// SIMATIC STEP 7 (V5.x) project COB#1&2_EL#2_01_07_2014
// CPU: CPU 315-2 DP
// CPU: CPU 315-2 DP

SYMBOL_TABLE
"FWD_END_POSI"	DB 1	DB 1	// FWD END POSITION LIMIT SWITCH
"OUTPUT_MAPPING_DB"	DB 2	DB 2	// TRAVEL DELAY TIME
"TRAVEL_DRIVE_DB"	DB 3	DB 3	// QUNCHING START PB
"COMMON_DB"	DB 4	DB 4
"TATA_COMMUNICATION_DB"	DB 5	DB 5	// TATA COMMUNIATION DATA BLOCK
"WinCC_Interface_DB"	DB 6	DB 6
"POWER_ON_DB"	DB 7	DB 7
"ACTUAL_TIME_DB"	DB 8	DB 8
"COMPRESSOR_DB"	DB 9	DB 9
"PROFIBUS_DATA"	DB 10	DB 10
"CMD_FROM_TATA"	DB 11	DB 11	// COMMANDS FROM TATA THROUGH PROFIBUS
"FB_TO_TATA"	DB 12	DB 12	// FEEDBACK TO TATA THROUGH PROFIBUS
"FLAPPER_GATE_DB"	DB 13	DB 13	// FLAPPER GATE DATA BLOCK
"RECEIVE_DB_342-5"	DB 21	DB 21
"SEND_DB_342-5"	DB 22	DB 22
"SPARE_1_DB"	DB 89	DB 89
"SPARE_2_DB"	DB 90	DB 90
"TDISCON"	FB 66	FB 66	// Disconnect
"POWER ON"	FC 2	FC 2	// MAIN POWER ON
"COMPRESSOR"	FC 3	FC 3
"FLAPPER_GATE"	FC 4	FC 4	// FLAPPER GATE FEEDBACKS
"ALARMS"	FC 5	FC 5
"INPUT_MAPPING"	FC 6	FC 6
"OUTPUT_MAPPING"	FC 7	FC 7
"TRAVEL_DRIVE_PROFI_MODE"	FC 8	FC 8
"TRAVEL_DRIVE"	FC 9	FC 9	// TRAVEL DRIVE IN HARDWARE AND PROFIBUS MODES
"PROFIBUS_COMMUNICATION"	FC 10	FC 10	// PROFIBUS COMMUNICATION
"TATA_COMMUNICATION"	FC 11	FC 11	// COMMUNICATION WITH TATA THROUGH PROFIBUS
"FAULT TRAP"	FC 12	FC 12	// FAULT EXAMINATION FC
"SCALE"	FC 105	FC 105	// Scaling Values
"UNSCALE"	FC 106	FC 106	// Unscaling Values
"MAIN PWR RUNG FB"	I 0.0	BOOL	// MAIN POWER RUNNING FEEDBACK
"CONTROL PWR ON FB"	I 0.1	BOOL	// CONTROL POWER ON FEEDBACK
"EMER STOP PB AT CD"	I 0.2	BOOL	// EMERGENCY STOP PUSH BUTTON AT CD
"LAMP TEST PB ATCD"	I 0.3	BOOL	// LAMP TEST PUSH BUTTON AT CD
"ALARM ACK PB AT CD"	I 0.4	BOOL	// ALARM ACKNOWLEDGE PUSH BUTTON AT CD
"MANUAL MODE"	I 0.5	BOOL	// MANUAL MODE SELECTION
"AUTO MODE"	I 0.6	BOOL	// AUTO MODE SELECTION
"LT_CRIPPING_SPEED"	I 0.7	BOOL	// LT TRAVEL CRIPPING SPEED
"PROFIBUS/HW DRV1 SELCT"	I 1.0	BOOL	// PROFIBUS/HARDWARE MODE SELECT DRIVE 1
"TRVL DRV 1 RDY TO START"	I 1.1	BOOL	// TRAVEL DRIVE 1 READY TO START
"TRVL DRV 1 RNG FB"	I 1.2	BOOL	// TRAVEL DRIVE 1 RUNNING FEED BACK
"TRVL DRV 1 OLR TRIP"	I 1.3	BOOL	// TRAVEL DRIVE 1 OLR TRIPPED FEED BACK
"PROFIBUS/HW DRV2 SELCT"	I 1.4	BOOL	// PROFIBUS/HARDWARE MODE SELECT DRIVE 2
"TRVL DRV 2 RDY TO START"	I 1.5	BOOL	// TRAVEL DRIVE 2 READY TO START
"TRVL DRV 2 RNG FB"	I 1.6	BOOL	// TRAVEL DRIVE 2 RUNNING FEED BACK
"TRVL DRV 2 OLR TRIP"	I 1.7	BOOL	// TRAVEL DRIVE 2 OLR TRIPPED FEED BACK
"SPARE _2"	I 2.0	BOOL	// SPARE 2
"SPARE_3"	I 2.1	BOOL	// SPARE_3
"JOY ST DEADMAN BUTTON"	I 2.2	BOOL	// JOYSTICK DEADMAN BUTTON
"JOY ST HOME POS"	I 2.3	BOOL	// JOYSTICK HOME POSITION
"JOY ST FWD POS"	I 2.4	BOOL	// JOYSTICK FORWARD POSITION
"JOY ST REV POS"	I 2.5	BOOL	// JOYSTICK REVERSE POSITION
"EMER STOP AT MCC"	I 2.6	BOOL	// EMERGENCY STOP PUSH BUTTON AT MCC
"QL_NOT_RDY_INPUT"	I 2.7	BOOL	// QUENCHING NOT READY
"FWD END LMT SW FB"	I 3.0	BOOL	// FORWARD END LIMIT SWITCH FEED BACK
"FWD EMER END LMT SW FB"	I 3.1	BOOL	// FORWARD EMERGENCY END LIMIT SWITCH FEED BACK
"REV END LMT SW FB"	I 3.2	BOOL	// REVERSE END LIMIT SWITCH FEED BACK
"REV EMER END LMT SW FB"	I 3.3	BOOL	// REVERSE EMERGENCY END LIMIT SWITCH FEED BACK
"LS_FLAPPER_GATE_1_FB"	I 3.4	BOOL	// LS_FLAPPER_GATE 1 FB
"LS_FLAPPER_GATE_2_FB"	I 3.5	BOOL	// LS FLAPPER GATE 2 FB
"DRIVE_1_ISU_CHARGE"	I 3.6	BOOL	// DRIVE 1 ISU CHARGE
"DRIVE_2_ISU_CHARGE"	I 3.7	BOOL	// DRIVE 2 ISU CHARGE
"COMP 1 RDY TO START"	I 4.0	BOOL	// COMPRESSOR 1 READY TO START PUSH BUTTON
"COMP1 RUNG FB"	I 4.1	BOOL	// COMPRESSOR 1 RUNNING FEED BACK
"COMP 2 RDY TO START"	I 4.2	BOOL	// COMPRESSOR 2 READY TO START PUSH BUTTON
"COMP2 RUNG FB"	I 4.3	BOOL	// COMPRESSOR 2 RUNNING FEED BACK
"COMP 1 & 2 SELECT"	I 4.4	BOOL	// COMPRESSOR 1 & 2 SELECTION
"COMP 1 START PB"	I 4.5	BOOL	// COMPRESSOR 1 START PUSH BUTTON
"COMP 1 STOP PB"	I 4.6	BOOL	// COMPRESSOR 1 STOP PUSH BUTTON
"CD_PC_SEL"	I 4.7	BOOL	// CD OR PC SELECTION SWITCH
"COMP 2 START PB"	I 5.0	BOOL	// COMPRESSOR 2 START PUSH BUTTON
"COMP 2 STOP PB"	I 5.1	BOOL	// COMPRESSOR 2 STOP PUSH BUTTON
"COMP1 MAX PSW FB"	I 5.2	BOOL	// COMPRESSOR 1 MAX PRESSURE SWITCH FEED BACK
"COMP MINI PSW FB"	I 5.3	BOOL	// MINIMUM PRESSURE SWITCH FEED BACK TRAVEL
"COMP BRK LINE PSW FB"	I 5.4	BOOL	// LT BRAKE LINE PRESSURE SWITCH FEED BACK
"COMP2 CNTRL PSW FB"	I 5.5	BOOL	// COMPRESSOR 2 CONTROL PRESSURE SWITCH FEED BACK
"SPARE 4"	I 5.6	BOOL	// SPARE INPUT 4 (I5.6)
"SPARE 5"	I 5.7	BOOL	// SPARE INPUT 5 (I5.7)
"SPARE 6"	I 6.0	BOOL	// SPARE INPUT 6 (I6.0)
"PUSHING_PERMISION"	I 6.1	BOOL	// PUSHING PERMISSION SIGNAL
"FED_END_POSI"	I 6.2	BOOL	// FWD END POSITION LIMIT SWITCH
"SPARE 9"	I 6.3	BOOL	// SPARE INPUT 9 (I6.3)
"SPARE 10"	I 6.4	BOOL	// SPARE INPUT 10 (I6.4)
"SPARE 11"	I 6.5	BOOL	// SPARE INPUT 11 (I6.5)
"SPARE 12"	I 6.6	BOOL	// SPARE INPUT 12 (I6.6)
"SPARE 13"	I 6.7	BOOL	// SPARE INPUT 13 (I6.7)
"SPARE 14"	I 7.0	BOOL	// SPARE INPUT 14 (I7.0)
"SPARE 15"	I 7.1	BOOL	// SPARE INPUT 15 (I7.1)
"SPARE 16"	I 7.2	BOOL	// SPARE INPUT 16 (I7.2)
"SPARE 17"	I 7.3	BOOL	// SPARE INPUT 17 (I7.3)
"SPARE 18"	I 7.4	BOOL	// SPARE INPUT 18 (I7.4)
"SPARE 19"	I 7.5	BOOL	// SPARE INPUT 19 (I7.5)
"SPARE 20"	I 7.6	BOOL	// SPARE INPUT 20 (I7.6)
"SPARE 21"	I 7.7	BOOL	// SPARE INPUT 21 (I7.7)
"LOW BIT"	M 0.0	BOOL	// ALWAYS LOW BIT
"HIGH BIT"	M 0.1	BOOL	// ALWAYS HIGH BIT
"QUENCHING_INPUT_LS"	M 2.0	BOOL
"40S_LT_ON_DELAY"	M 2.1	BOOL	// 40 SECOND LT ON DELAY
"QUEN_DELEY_TIME"	M 2.2	BOOL	// QIENCHING DELAY OFF TIME
"LT_PERMISSION"	M 2.3	BOOL	// LT  AFTER QUENCHING PERMISSION
"COMP_1_RDY_2_STRT_FLT"	M 2.4	BOOL	// COMP#1 READY TO START FEEDBACK FAULT
"EMER_CD_FLT"	M 2.5	BOOL	// EMERGENCY AT CD FAULT
"COMP_1_STP_PB_FLT"	M 2.6	BOOL	// COMP#1 STOP PUSH BUTTON FAULT
"COMP_2_RDY_FR_STRT_FLT"	M 2.7	BOOL	// COMPRESSOR 2 READY FOR START FAULT
"COMP_2_OFF_PB_FLT"	M 3.0	BOOL	// COMPRESSOR 2 OFF PUSH BUTTON FAULT
"RESET FAULTS"	M 3.1	BOOL	// RESET ALL FAULTS
"COMP_SELEC_SW_FLT"	M 3.2	BOOL	// COMPRESSOR SELECTOR SWITCH FAULT
"MAIN_PWR_FLT"	M 3.3	BOOL	// MAIN POWER ON FEEDBACK FAULT
"CTRL_PWR_FLT"	M 3.4	BOOL	// CONTROL POWER ON FEEDBACK FAULT
"CYCLIC_EXECUCTION"	OB 1	OB 1	// Cycle Execution
"CYCL_FLT"	OB 80	OB 80	// Cycle Time Fault
"I/O_FLT1"	OB 82	OB 82	// I/O Point Fault 1
"OBNL_FLT"	OB 85	OB 85	// OB Not Loaded Fault
"RACK_FLT"	OB 86	OB 86	// Loss of Rack Fault
"COMM_FLT"	OB 87	OB 87	// Communication Fault
"COMPLETE RESTART"	OB 100	OB 100	// Complete Restart
"PROG_ERR"	OB 121	OB 121	// Programming Error
"MOD_ERR"	OB 122	OB 122	// Module Access Error
"JOY_STICK_SPEED_REF"	PIW 254	INT	// SPEED REFERENCE FROM JOY STICK
"SPEED_REF_TO_DRV_1"	PQW 258	INT	// SPEED REFERENCE TO TRAVEL DRIVE 1
"SPEED_REF_TO_DRV_2"	PQW 260	INT	// SPEED REFERENCE TO TRAVEL DRIVE 2
"CNTRL_ PWR_ ON_ IND"	Q 0.2	BOOL	// CONTROL POWER ON INDICATION
"COMP_ 1_ON_CMD"	Q 0.3	BOOL	// COMPRESSOR-1 ON COMMAND
"COMP_ 2_ON_CMD"	Q 0.4	BOOL	// COMPRESSOR 2 ON COMMAND
"FLAPPER_GATE_1_POSITION"	Q 0.5	BOOL	// FLAPPER_GATE_1_POSITION
"FLAPPER_GATE_2_POSITION"	Q 0.6	BOOL	// "FLAPPER_GATE_2_POSITION"
"FLAP_GATE_1_OPN_IND"	Q 0.7	BOOL	// FLAPPER GATE 1 OPEN INDICATION
"TRA_DRIVE_1_FWD_COM"	Q 1.0	BOOL	// TRAVEL DRIVE 1 FORWARD COMMAND
"TRA_DRIVE_1_REV_COM"	Q 1.1	BOOL	// TRAVEL DRIVE 1 REVERSE COMMAND
"TRA_DRIVE_2_FWD_COM"	Q 1.2	BOOL	// TRAVEL DRIVE 2 FORWRD COMMAND
"TRA_DRIVE_2_REV_COM"	Q 1.3	BOOL	// TRAVEL DRIVE 2 REVERSE COMMAND
"COM_1_ON_IND"	Q 1.4	BOOL	// COMPRESSOR 1 ON INDICATION
"COM_2_ON_IND"	Q 1.5	BOOL	// COMPRESSOR 2 ON INDICATION
"TRA_PERMISSION_IND"	Q 1.6	BOOL	// TRAVEL PERMISSION INDICATION
"FLAP_GATE_2_OPN_IND"	Q 1.7	BOOL	// FLAPPER GATE 2 OPEN INDICATION
"DRV_1_ISU_CMD"	Q 2.0	BOOL	// DRIVE 1 ISU CHARGE COMMAND
"DRV_2_ISU_CMD"	Q 2.1	BOOL	// DRIVE 2 ISU CHARGE COMMAND
"LIGHT_ON_CMD"	Q 2.2	BOOL	// LIGHT ON COMMAND
"SPARE_12"	Q 2.3	BOOL	// SPARE_12
"SPARE OP 9"	Q 2.4	BOOL	// SPARE OUPUT 1 (Q2.4)
"SPARE OP 10"	Q 2.5	BOOL	// TRAVEL DELAY TIME (Q2.5)
"SPARE OP 11"	Q 2.6	BOOL	// SPARE OUPUT 1 (Q2.6)
"SPARE OP 12"	Q 2.7	BOOL	// SPARE OUPUT 1 (Q2.7)
"SPARE OP 13"	Q 3.0	BOOL	// SPARE OUPUT 1 (Q3.0)
"SPARE OP 14"	Q 3.1	BOOL	// SPARE OUPUT 1 (Q3.1)
"SPARE OP 15"	Q 3.2	BOOL	// SPARE OUPUT 1 (Q3.2)
"SPARE OP 16"	Q 3.3	BOOL	// SPARE OUPUT 1 (Q3.3)
"SPARE OP 17"	Q 3.4	BOOL	// SPARE OUPUT 1 (Q3.4)
"SPARE OP 18"	Q 3.5	BOOL	// SPARE OUPUT 1 (Q3.5)
"SPARE OP 19"	Q 3.6	BOOL	// SPARE OUPUT 1 (Q3.6)
"SPARE OP 20"	Q 3.7	BOOL	// SPARE OUPUT 1 (Q3.7)
"HOOTER_ON_OP"	Q 4.0	BOOL	// HOOTER ON OUTPUT
"DPRD_DAT"	SFC 14	SFC 14	// Read Consistent Data of a Standard DP Slave
"DPWR_DAT"	SFC 15	SFC 15	// Write Consistent Data to a Standard DP Slave
"VAT_1"	VAT 1	
"FAULT_EXAMINATION"	VAT 2		// FAULT EXAMINATION TABLE
"LOCO#2_FORCE TABLE"	VAT 3	
END_SYMBOL_TABLE

// FB 66: know-how protected block, not included

FUNCTION "POWER ON" : VOID	// FC 2
VERSION : 0.1
VAR_TEMP
  TEMP0 : WORD ;
  TEMP1 : WORD ;
  TEMP2 : WORD ;
END_VAR
BEGIN
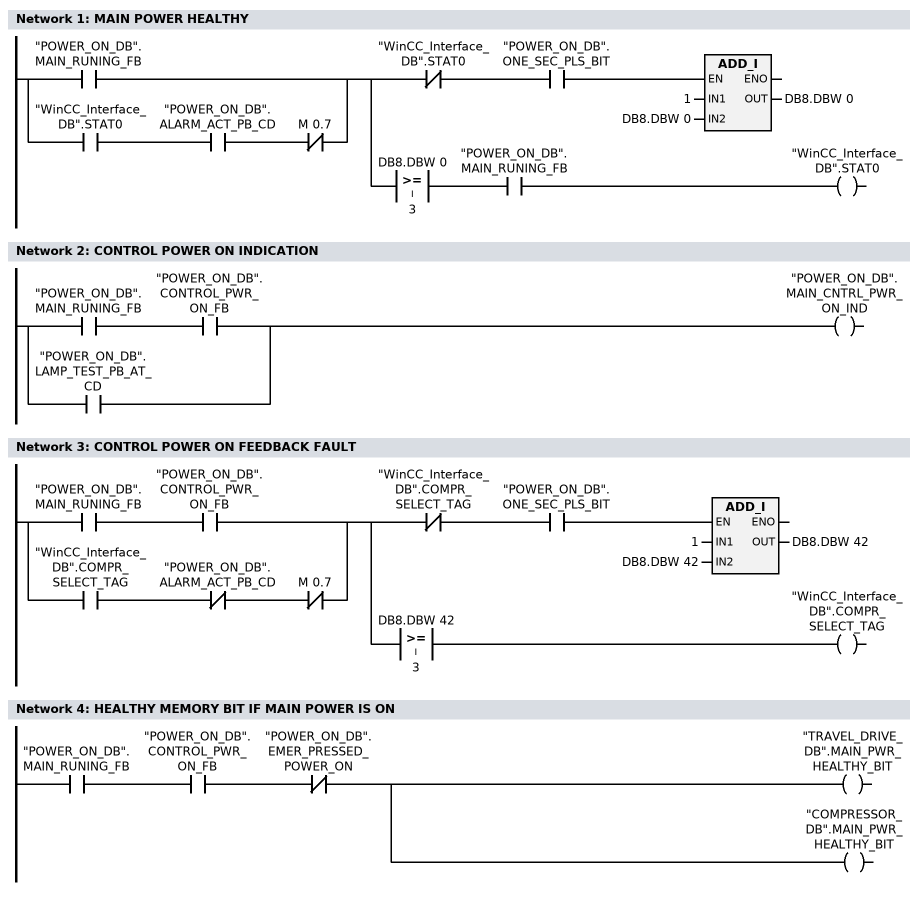
NETWORK
TITLE = MAIN POWER HEALTHY
      O     "POWER_ON_DB".MAIN_RUNING_FB;
      O;
      A     "WinCC_Interface_DB".STAT0;
      A     "POWER_ON_DB".ALARM_ACT_PB_CD;
      AN    M 0.7;
      =     L 6.0;
      A     L 6.0;
      AN    "WinCC_Interface_DB".STAT0;
      A     "POWER_ON_DB".ONE_SEC_PLS_BIT;
      JNB   _001;
      L     1;
      L     DB8.DBW 0;
      +I;
      T     DB8.DBW 0;
_001: NOP   0;
      A     L 6.0;
      A(;
      L     DB8.DBW 0;
      L     3;
      >=I;
      );
      A     "POWER_ON_DB".MAIN_RUNING_FB;
      =     "WinCC_Interface_DB".STAT0;
NETWORK
TITLE = CONTROL POWER ON INDICATION
      A     "POWER_ON_DB".MAIN_RUNING_FB;
      A     "POWER_ON_DB".CONTROL_PWR_ON_FB;
      O     "POWER_ON_DB".LAMP_TEST_PB_AT_CD;
      =     "POWER_ON_DB".MAIN_CNTRL_PWR_ON_IND;
NETWORK
TITLE = CONTROL POWER ON FEEDBACK FAULT
      A     "POWER_ON_DB".MAIN_RUNING_FB;
      A     "POWER_ON_DB".CONTROL_PWR_ON_FB;
      O;
      A     "WinCC_Interface_DB".COMPR_SELECT_TAG;
      AN    "POWER_ON_DB".ALARM_ACT_PB_CD;
      AN    M 0.7;
      =     L 6.0;
      A     L 6.0;
      AN    "WinCC_Interface_DB".COMPR_SELECT_TAG;
      A     "POWER_ON_DB".ONE_SEC_PLS_BIT;
      JNB   _002;
      L     1;
      L     DB8.DBW 42;
      +I;
      T     DB8.DBW 42;
_002: NOP   0;
      A     L 6.0;
      A(;
      L     DB8.DBW 42;
      L     3;
      >=I;
      );
      =     "WinCC_Interface_DB".COMPR_SELECT_TAG;
NETWORK
TITLE = HEALTHY MEMORY BIT IF MAIN POWER IS ON
      A     "POWER_ON_DB".MAIN_RUNING_FB;
      A     "POWER_ON_DB".CONTROL_PWR_ON_FB;
      AN    "POWER_ON_DB".EMER_PRESSED_POWER_ON;
      =     "TRAVEL_DRIVE_DB".MAIN_PWR_HEALTHY_BIT;
      =     "COMPRESSOR_DB".MAIN_PWR_HEALTHY_BIT;
END_FUNCTION

FUNCTION "COMPRESSOR" : VOID	// FC 3
VERSION : 0.1
BEGIN
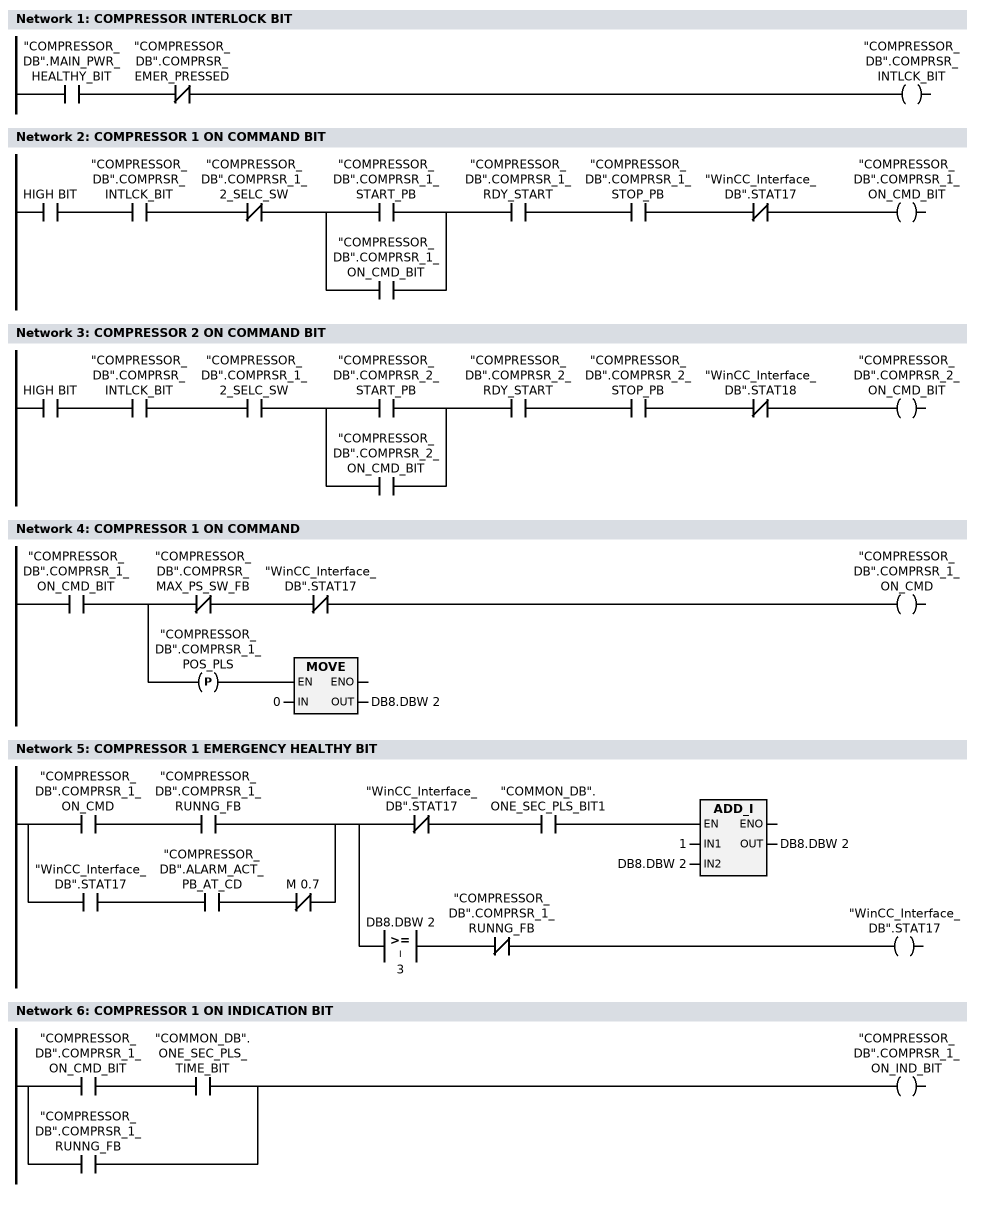
NETWORK
TITLE = COMPRESSOR INTERLOCK BIT
      A     "COMPRESSOR_DB".MAIN_PWR_HEALTHY_BIT;
      AN    "COMPRESSOR_DB".COMPRSR_EMER_PRESSED;
      =     "COMPRESSOR_DB".COMPRSR_INTLCK_BIT;
NETWORK
TITLE = COMPRESSOR 1 ON COMMAND BIT
      A     "HIGH BIT";
      A     "COMPRESSOR_DB".COMPRSR_INTLCK_BIT;
      AN    "COMPRESSOR_DB".COMPRSR_1_2_SELC_SW;
      A(;
      O     "COMPRESSOR_DB".COMPRSR_1_START_PB;
      O     "COMPRESSOR_DB".COMPRSR_1_ON_CMD_BIT;
      );
      A     "COMPRESSOR_DB".COMPRSR_1_RDY_START;
      A     "COMPRESSOR_DB".COMPRSR_1_STOP_PB;
      AN    "WinCC_Interface_DB".STAT17;
      =     "COMPRESSOR_DB".COMPRSR_1_ON_CMD_BIT;
NETWORK
TITLE = COMPRESSOR 2 ON COMMAND BIT
      A     "HIGH BIT";
      A     "COMPRESSOR_DB".COMPRSR_INTLCK_BIT;
      A     "COMPRESSOR_DB".COMPRSR_1_2_SELC_SW;
      A(;
      O     "COMPRESSOR_DB".COMPRSR_2_START_PB;
      O     "COMPRESSOR_DB".COMPRSR_2_ON_CMD_BIT;
      );
      A     "COMPRESSOR_DB".COMPRSR_2_RDY_START;
      A     "COMPRESSOR_DB".COMPRSR_2_STOP_PB;
      AN    "WinCC_Interface_DB".STAT18;
      =     "COMPRESSOR_DB".COMPRSR_2_ON_CMD_BIT;
NETWORK
TITLE = COMPRESSOR 1 ON COMMAND
      A     "COMPRESSOR_DB".COMPRSR_1_ON_CMD_BIT;
      =     L 0.0;
      A     L 0.0;
      AN    "COMPRESSOR_DB".COMPRSR_MAX_PS_SW_FB;
      AN    "WinCC_Interface_DB".STAT17;
      =     "COMPRESSOR_DB".COMPRSR_1_ON_CMD;
      A     L 0.0;
      FP    "COMPRESSOR_DB".COMPRSR_1_POS_PLS;
      JNB   _001;
      L     0;
      T     DB8.DBW 2;
_001: NOP   0;
NETWORK
TITLE = COMPRESSOR 1 EMERGENCY HEALTHY BIT
      A     "COMPRESSOR_DB".COMPRSR_1_ON_CMD;
      A     "COMPRESSOR_DB".COMPRSR_1_RUNNG_FB;
      O;
      A     "WinCC_Interface_DB".STAT17;
      A     "COMPRESSOR_DB".ALARM_ACT_PB_AT_CD;
      AN    M 0.7;
      =     L 0.0;
      A     L 0.0;
      AN    "WinCC_Interface_DB".STAT17;
      A     "COMMON_DB".ONE_SEC_PLS_BIT1;
      JNB   _002;
      L     1;
      L     DB8.DBW 2;
      +I;
      T     DB8.DBW 2;
_002: NOP   0;
      A     L 0.0;
      A(;
      L     DB8.DBW 2;
      L     3;
      >=I;
      );
      AN    "COMPRESSOR_DB".COMPRSR_1_RUNNG_FB;
      =     "WinCC_Interface_DB".STAT17;
NETWORK
TITLE = COMPRESSOR 1 ON INDICATION BIT
      A     "COMPRESSOR_DB".COMPRSR_1_ON_CMD_BIT;
      A     "COMMON_DB".ONE_SEC_PLS_TIME_BIT;
      O     "COMPRESSOR_DB".COMPRSR_1_RUNNG_FB;
      =     "COMPRESSOR_DB".COMPRSR_1_ON_IND_BIT;
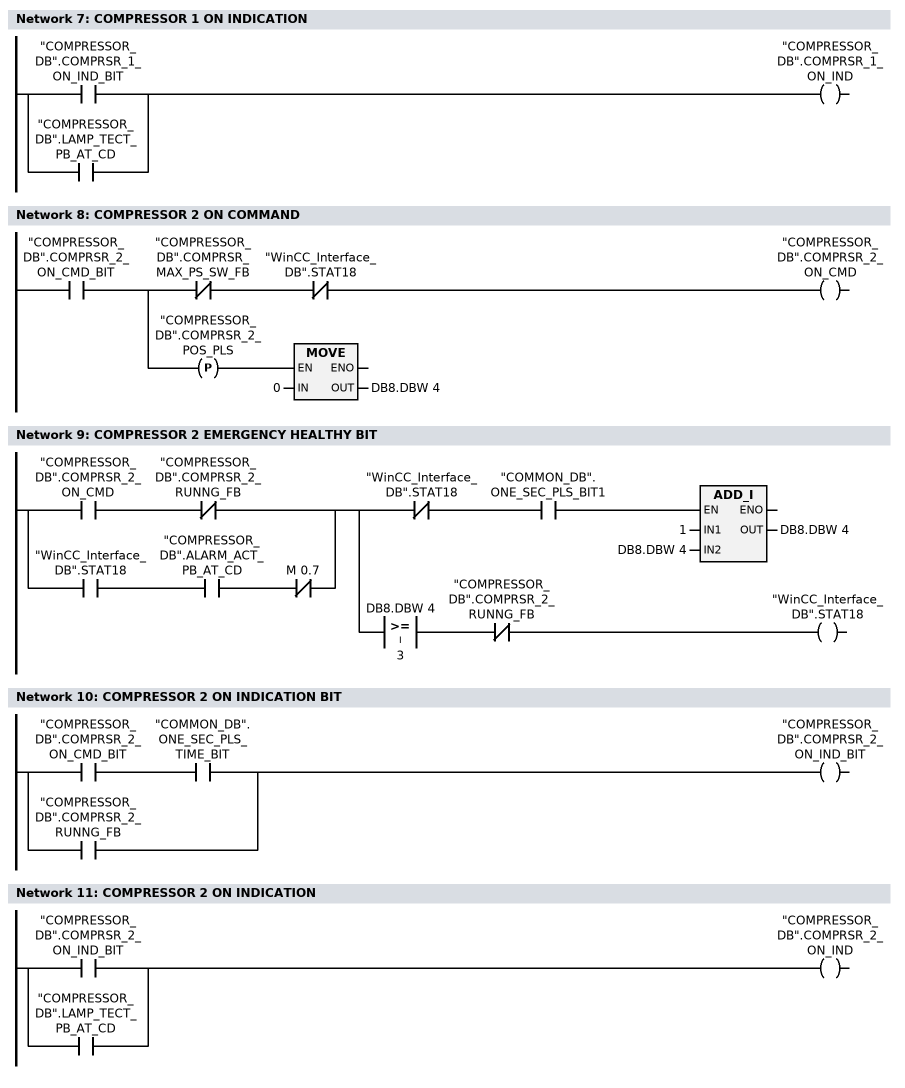
NETWORK
TITLE = COMPRESSOR 1 ON INDICATION
      O     "COMPRESSOR_DB".COMPRSR_1_ON_IND_BIT;
      O     "COMPRESSOR_DB".LAMP_TECT_PB_AT_CD;
      =     "COMPRESSOR_DB".COMPRSR_1_ON_IND;
NETWORK
TITLE = COMPRESSOR 2 ON COMMAND
      A     "COMPRESSOR_DB".COMPRSR_2_ON_CMD_BIT;
      =     L 0.0;
      A     L 0.0;
      AN    "COMPRESSOR_DB".COMPRSR_MAX_PS_SW_FB;
      AN    "WinCC_Interface_DB".STAT18;
      =     "COMPRESSOR_DB".COMPRSR_2_ON_CMD;
      A     L 0.0;
      FP    "COMPRESSOR_DB".COMPRSR_2_POS_PLS;
      JNB   _003;
      L     0;
      T     DB8.DBW 4;
_003: NOP   0;
NETWORK
TITLE = COMPRESSOR 2 EMERGENCY HEALTHY BIT
      A     "COMPRESSOR_DB".COMPRSR_2_ON_CMD;
      AN    "COMPRESSOR_DB".COMPRSR_2_RUNNG_FB;
      O;
      A     "WinCC_Interface_DB".STAT18;
      A     "COMPRESSOR_DB".ALARM_ACT_PB_AT_CD;
      AN    M 0.7;
      =     L 0.0;
      A     L 0.0;
      AN    "WinCC_Interface_DB".STAT18;
      A     "COMMON_DB".ONE_SEC_PLS_BIT1;
      JNB   _004;
      L     1;
      L     DB8.DBW 4;
      +I;
      T     DB8.DBW 4;
_004: NOP   0;
      A     L 0.0;
      A(;
      L     DB8.DBW 4;
      L     3;
      >=I;
      );
      AN    "COMPRESSOR_DB".COMPRSR_2_RUNNG_FB;
      =     "WinCC_Interface_DB".STAT18;
NETWORK
TITLE = COMPRESSOR 2 ON INDICATION BIT
      A     "COMPRESSOR_DB".COMPRSR_2_ON_CMD_BIT;
      A     "COMMON_DB".ONE_SEC_PLS_TIME_BIT;
      O     "COMPRESSOR_DB".COMPRSR_2_RUNNG_FB;
      =     "COMPRESSOR_DB".COMPRSR_2_ON_IND_BIT;
NETWORK
TITLE = COMPRESSOR 2 ON INDICATION
      O     "COMPRESSOR_DB".COMPRSR_2_ON_IND_BIT;
      O     "COMPRESSOR_DB".LAMP_TECT_PB_AT_CD;
      =     "COMPRESSOR_DB".COMPRSR_2_ON_IND;
END_FUNCTION

FUNCTION "FLAPPER_GATE" : VOID	// FC 4
VERSION : 0.1
BEGIN
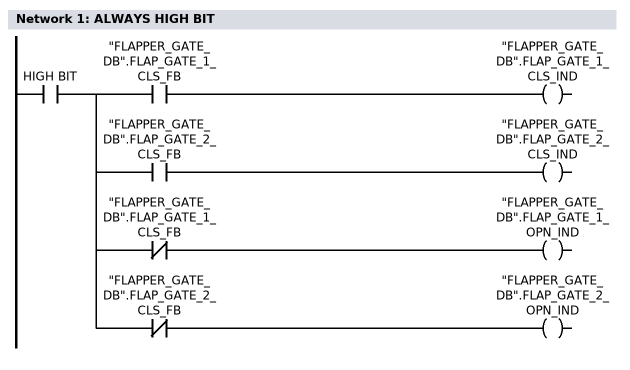
NETWORK
TITLE = ALWAYS HIGH BIT
      A     "HIGH BIT";
      =     L 0.0;
      A     L 0.0;
      A     "FLAPPER_GATE_DB".FLAP_GATE_1_CLS_FB;
      =     "FLAPPER_GATE_DB".FLAP_GATE_1_CLS_IND;
      A     L 0.0;
      A     "FLAPPER_GATE_DB".FLAP_GATE_2_CLS_FB;
      =     "FLAPPER_GATE_DB".FLAP_GATE_2_CLS_IND;
      A     L 0.0;
      AN    "FLAPPER_GATE_DB".FLAP_GATE_1_CLS_FB;
      =     "FLAPPER_GATE_DB".FLAP_GATE_1_OPN_IND;
      A     L 0.0;
      AN    "FLAPPER_GATE_DB".FLAP_GATE_2_CLS_FB;
      =     "FLAPPER_GATE_DB".FLAP_GATE_2_OPN_IND;
END_FUNCTION

FUNCTION "ALARMS" : VOID	// FC 5
VERSION : 0.1
BEGIN
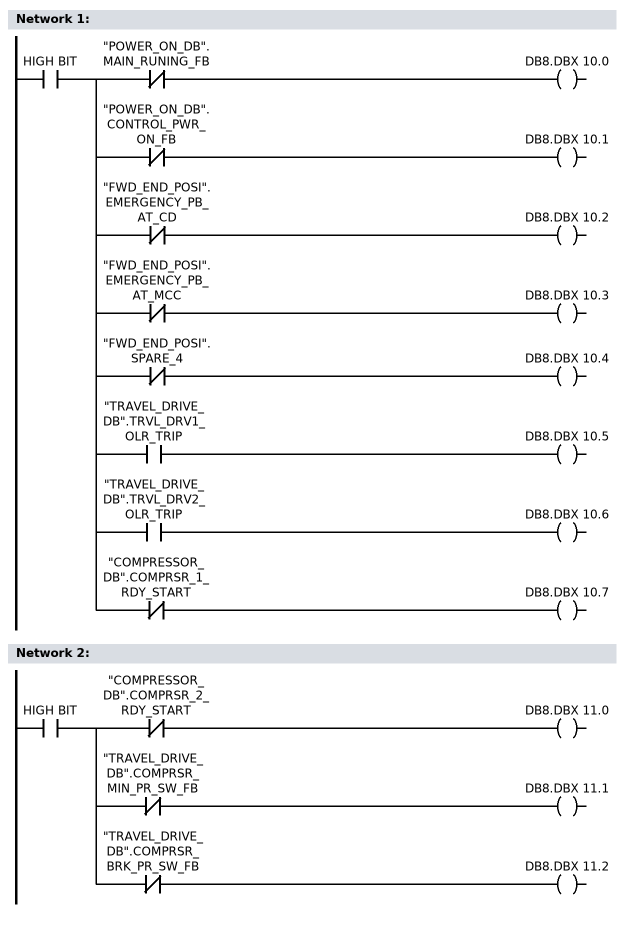
NETWORK
TITLE =
      A     "HIGH BIT";
      =     L 0.0;
      A     L 0.0;
      AN    "POWER_ON_DB".MAIN_RUNING_FB;
      =     DB8.DBX 10.0;
      A     L 0.0;
      AN    "POWER_ON_DB".CONTROL_PWR_ON_FB;
      =     DB8.DBX 10.1;
      A     L 0.0;
      AN    "FWD_END_POSI".EMERGENCY_PB_AT_CD;
      =     DB8.DBX 10.2;
      A     L 0.0;
      AN    "FWD_END_POSI".EMERGENCY_PB_AT_MCC;
      =     DB8.DBX 10.3;
      A     L 0.0;
      AN    "FWD_END_POSI".SPARE_4;
      =     DB8.DBX 10.4;
      A     L 0.0;
      A     "TRAVEL_DRIVE_DB".TRVL_DRV1_OLR_TRIP;
      =     DB8.DBX 10.5;
      A     L 0.0;
      A     "TRAVEL_DRIVE_DB".TRVL_DRV2_OLR_TRIP;
      =     DB8.DBX 10.6;
      A     L 0.0;
      AN    "COMPRESSOR_DB".COMPRSR_1_RDY_START;
      =     DB8.DBX 10.7;
NETWORK
TITLE =
      A     "HIGH BIT";
      =     L 0.0;
      A     L 0.0;
      AN    "COMPRESSOR_DB".COMPRSR_2_RDY_START;
      =     DB8.DBX 11.0;
      A     L 0.0;
      AN    "TRAVEL_DRIVE_DB".COMPRSR_MIN_PR_SW_FB;
      =     DB8.DBX 11.1;
      A     L 0.0;
      AN    "TRAVEL_DRIVE_DB".COMPRSR_BRK_PR_SW_FB;
      =     DB8.DBX 11.2;
END_FUNCTION

FUNCTION "INPUT_MAPPING" : VOID	// FC 6
VERSION : 0.1
BEGIN
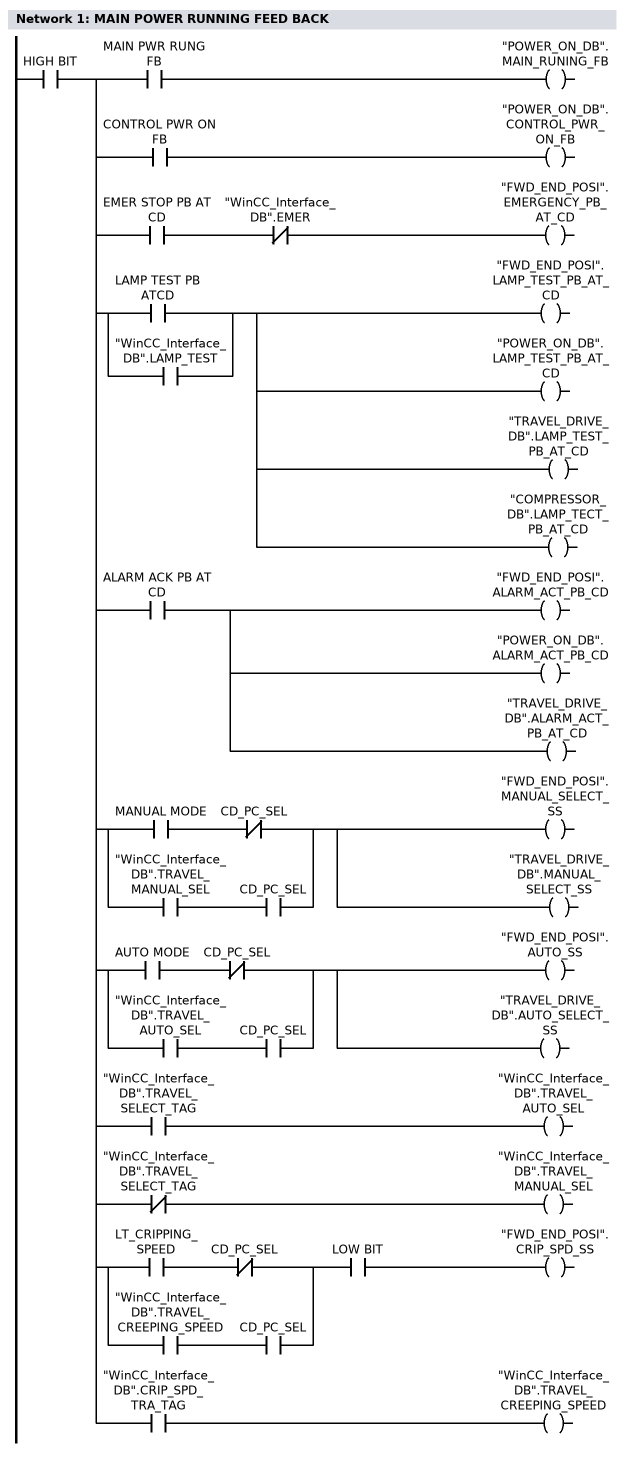
NETWORK
TITLE = MAIN POWER RUNNING FEED BACK
      A     "HIGH BIT";
      =     L 0.0;
      A     L 0.0;
      A     "MAIN PWR RUNG FB";
      =     "POWER_ON_DB".MAIN_RUNING_FB;
      A     L 0.0;
      A     "CONTROL PWR ON FB";
      =     "POWER_ON_DB".CONTROL_PWR_ON_FB;
      A     L 0.0;
      A     "EMER STOP PB AT CD";
      AN    "WinCC_Interface_DB".EMER;
      =     "FWD_END_POSI".EMERGENCY_PB_AT_CD;
      A     L 0.0;
      A(;
      O     "LAMP TEST PB ATCD";
      O     "WinCC_Interface_DB".LAMP_TEST;
      );
      =     "FWD_END_POSI".LAMP_TEST_PB_AT_CD;
      =     "POWER_ON_DB".LAMP_TEST_PB_AT_CD;
      =     "TRAVEL_DRIVE_DB".LAMP_TEST_PB_AT_CD;
      =     "COMPRESSOR_DB".LAMP_TECT_PB_AT_CD;
      A     L 0.0;
      A     "ALARM ACK PB AT CD";
      =     "FWD_END_POSI".ALARM_ACT_PB_CD;
      =     "POWER_ON_DB".ALARM_ACT_PB_CD;
      =     "TRAVEL_DRIVE_DB".ALARM_ACT_PB_AT_CD;
      A     L 0.0;
      A(;
      A     "MANUAL MODE";
      AN    "CD_PC_SEL";
      O;
      A     "WinCC_Interface_DB".TRAVEL_MANUAL_SEL;
      A     "CD_PC_SEL";
      );
      =     "FWD_END_POSI".MANUAL_SELECT_SS;
      =     "TRAVEL_DRIVE_DB".MANUAL_SELECT_SS;
      A     L 0.0;
      A(;
      A     "AUTO MODE";
      AN    "CD_PC_SEL";
      O;
      A     "WinCC_Interface_DB".TRAVEL_AUTO_SEL;
      A     "CD_PC_SEL";
      );
      =     "FWD_END_POSI".AUTO_SS;
      =     "TRAVEL_DRIVE_DB".AUTO_SELECT_SS;
      A     L 0.0;
      A     "WinCC_Interface_DB".TRAVEL_SELECT_TAG;
      =     "WinCC_Interface_DB".TRAVEL_AUTO_SEL;
      A     L 0.0;
      AN    "WinCC_Interface_DB".TRAVEL_SELECT_TAG;
      =     "WinCC_Interface_DB".TRAVEL_MANUAL_SEL;
      A     L 0.0;
      A(;
      A     "LT_CRIPPING_SPEED";
      AN    "CD_PC_SEL";
      O;
      A     "WinCC_Interface_DB".TRAVEL_CREEPING_SPEED;
      A     "CD_PC_SEL";
      );
      A     "LOW BIT";
      =     "FWD_END_POSI".CRIP_SPD_SS;
      A     L 0.0;
      A     "WinCC_Interface_DB".CRIP_SPD_TRA_TAG;
      =     "WinCC_Interface_DB".TRAVEL_CREEPING_SPEED;
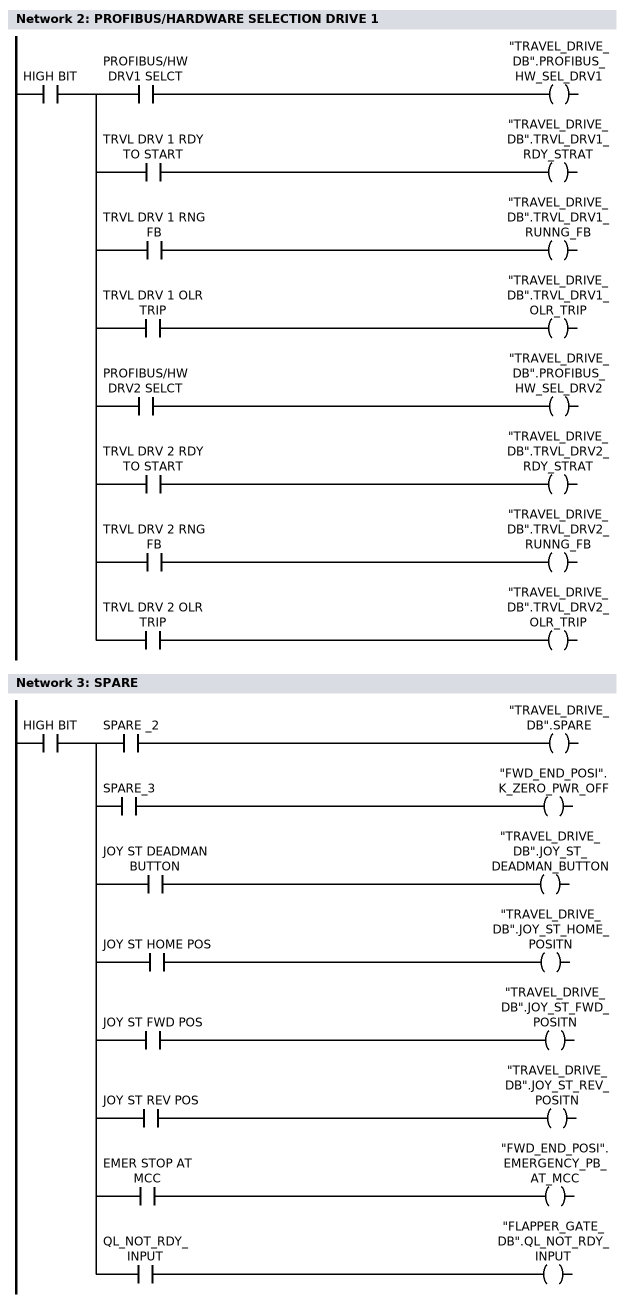
NETWORK
TITLE = PROFIBUS/HARDWARE SELECTION DRIVE 1
      A     "HIGH BIT";
      =     L 0.0;
      A     L 0.0;
      A     "PROFIBUS/HW DRV1 SELCT";
      =     "TRAVEL_DRIVE_DB".PROFIBUS_HW_SEL_DRV1;
      A     L 0.0;
      A     "TRVL DRV 1 RDY TO START";
      =     "TRAVEL_DRIVE_DB".TRVL_DRV1_RDY_STRAT;
      A     L 0.0;
      A     "TRVL DRV 1 RNG FB";
      =     "TRAVEL_DRIVE_DB".TRVL_DRV1_RUNNG_FB;
      A     L 0.0;
      A     "TRVL DRV 1 OLR TRIP";
      =     "TRAVEL_DRIVE_DB".TRVL_DRV1_OLR_TRIP;
      A     L 0.0;
      A     "PROFIBUS/HW DRV2 SELCT";
      =     "TRAVEL_DRIVE_DB".PROFIBUS_HW_SEL_DRV2;
      A     L 0.0;
      A     "TRVL DRV 2 RDY TO START";
      =     "TRAVEL_DRIVE_DB".TRVL_DRV2_RDY_STRAT;
      A     L 0.0;
      A     "TRVL DRV 2 RNG FB";
      =     "TRAVEL_DRIVE_DB".TRVL_DRV2_RUNNG_FB;
      A     L 0.0;
      A     "TRVL DRV 2 OLR TRIP";
      =     "TRAVEL_DRIVE_DB".TRVL_DRV2_OLR_TRIP;
NETWORK
TITLE = SPARE
//`
      A     "HIGH BIT";
      =     L 0.0;
      A     L 0.0;
      A     "SPARE _2";
      =     "TRAVEL_DRIVE_DB".SPARE;
      A     L 0.0;
      A     "SPARE_3";
      =     "FWD_END_POSI".K_ZERO_PWR_OFF;
      A     L 0.0;
      A     "JOY ST DEADMAN BUTTON";
      =     "TRAVEL_DRIVE_DB".JOY_ST_DEADMAN_BUTTON;
      A     L 0.0;
      A     "JOY ST HOME POS";
      =     "TRAVEL_DRIVE_DB".JOY_ST_HOME_POSITN;
      A     L 0.0;
      A     "JOY ST FWD POS";
      =     "TRAVEL_DRIVE_DB".JOY_ST_FWD_POSITN;
      A     L 0.0;
      A     "JOY ST REV POS";
      =     "TRAVEL_DRIVE_DB".JOY_ST_REV_POSITN;
      A     L 0.0;
      A     "EMER STOP AT MCC";
      =     "FWD_END_POSI".EMERGENCY_PB_AT_MCC;
      A     L 0.0;
      A     "QL_NOT_RDY_INPUT";
      =     "FLAPPER_GATE_DB".QL_NOT_RDY_INPUT;
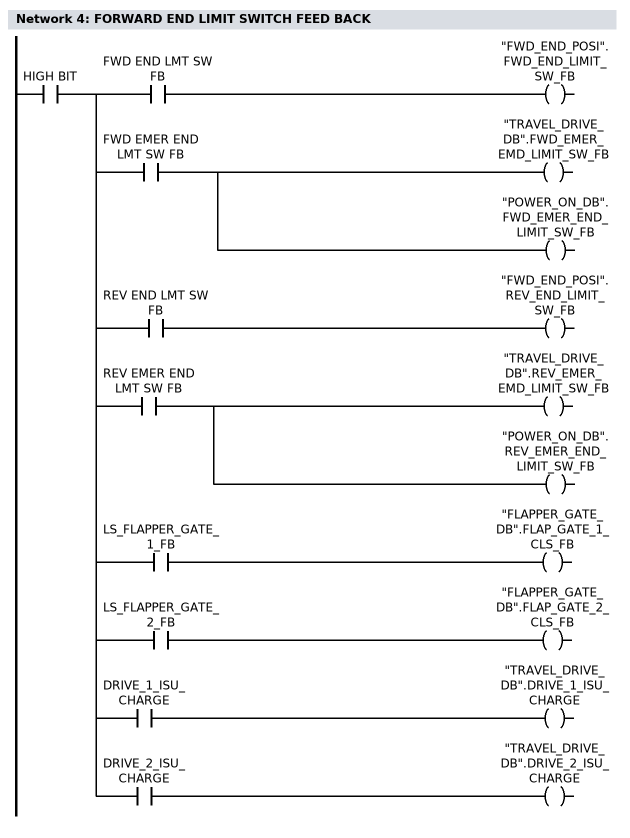
NETWORK
TITLE = FORWARD END LIMIT SWITCH FEED BACK
      A     "HIGH BIT";
      =     L 0.0;
      A     L 0.0;
      A     "FWD END LMT SW FB";
      =     "FWD_END_POSI".FWD_END_LIMIT_SW_FB;
      A     L 0.0;
      A     "FWD EMER END LMT SW FB";
      =     "TRAVEL_DRIVE_DB".FWD_EMER_EMD_LIMIT_SW_FB;
      =     "POWER_ON_DB".FWD_EMER_END_LIMIT_SW_FB;
      A     L 0.0;
      A     "REV END LMT SW FB";
      =     "FWD_END_POSI".REV_END_LIMIT_SW_FB;
      A     L 0.0;
      A     "REV EMER END LMT SW FB";
      =     "TRAVEL_DRIVE_DB".REV_EMER_EMD_LIMIT_SW_FB;
      =     "POWER_ON_DB".REV_EMER_END_LIMIT_SW_FB;
      A     L 0.0;
      A     "LS_FLAPPER_GATE_1_FB";
      =     "FLAPPER_GATE_DB".FLAP_GATE_1_CLS_FB;
      A     L 0.0;
      A     "LS_FLAPPER_GATE_2_FB";
      =     "FLAPPER_GATE_DB".FLAP_GATE_2_CLS_FB;
      A     L 0.0;
      A     "DRIVE_1_ISU_CHARGE";
      =     "TRAVEL_DRIVE_DB".DRIVE_1_ISU_CHARGE;
      A     L 0.0;
      A     "DRIVE_2_ISU_CHARGE";
      =     "TRAVEL_DRIVE_DB".DRIVE_2_ISU_CHARGE;
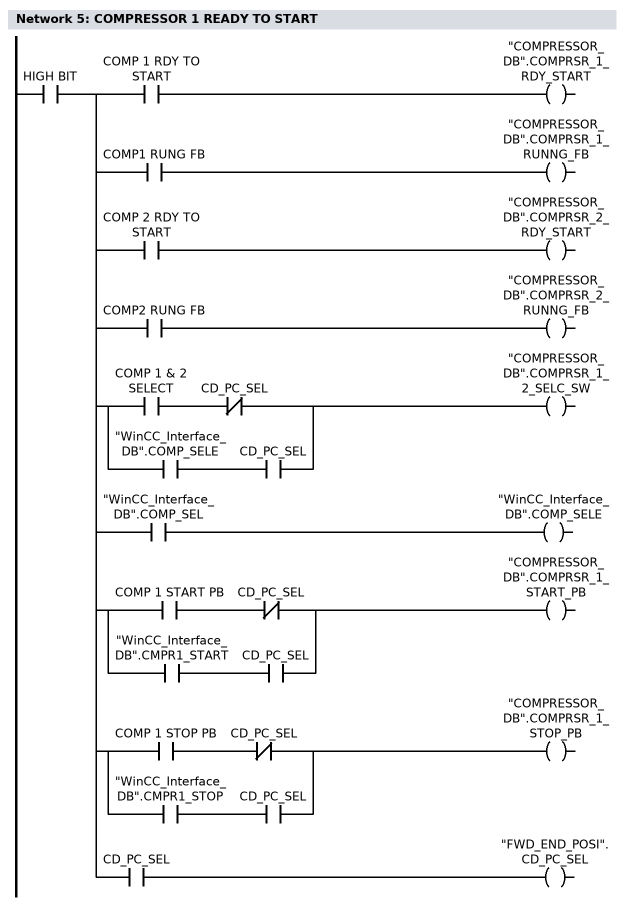
NETWORK
TITLE = COMPRESSOR 1 READY TO START
      A     "HIGH BIT";
      =     L 0.0;
      A     L 0.0;
      A     "COMP 1 RDY TO START";
      =     "COMPRESSOR_DB".COMPRSR_1_RDY_START;
      A     L 0.0;
      A     "COMP1 RUNG FB";
      =     "COMPRESSOR_DB".COMPRSR_1_RUNNG_FB;
      A     L 0.0;
      A     "COMP 2 RDY TO START";
      =     "COMPRESSOR_DB".COMPRSR_2_RDY_START;
      A     L 0.0;
      A     "COMP2 RUNG FB";
      =     "COMPRESSOR_DB".COMPRSR_2_RUNNG_FB;
      A     L 0.0;
      A(;
      A     "COMP 1 & 2 SELECT";
      AN    "CD_PC_SEL";
      O;
      A     "WinCC_Interface_DB".COMP_SELE;
      A     "CD_PC_SEL";
      );
      =     "COMPRESSOR_DB".COMPRSR_1_2_SELC_SW;
      A     L 0.0;
      A     "WinCC_Interface_DB".COMP_SEL;
      =     "WinCC_Interface_DB".COMP_SELE;
      A     L 0.0;
      A(;
      A     "COMP 1 START PB";
      AN    "CD_PC_SEL";
      O;
      A     "WinCC_Interface_DB".CMPR1_START;
      A     "CD_PC_SEL";
      );
      =     "COMPRESSOR_DB".COMPRSR_1_START_PB;
      A     L 0.0;
      A(;
      A     "COMP 1 STOP PB";
      AN    "CD_PC_SEL";
      O;
      A     "WinCC_Interface_DB".CMPR1_STOP;
      A     "CD_PC_SEL";
      );
      =     "COMPRESSOR_DB".COMPRSR_1_STOP_PB;
      A     L 0.0;
      A     "CD_PC_SEL";
      =     "FWD_END_POSI".CD_PC_SEL;
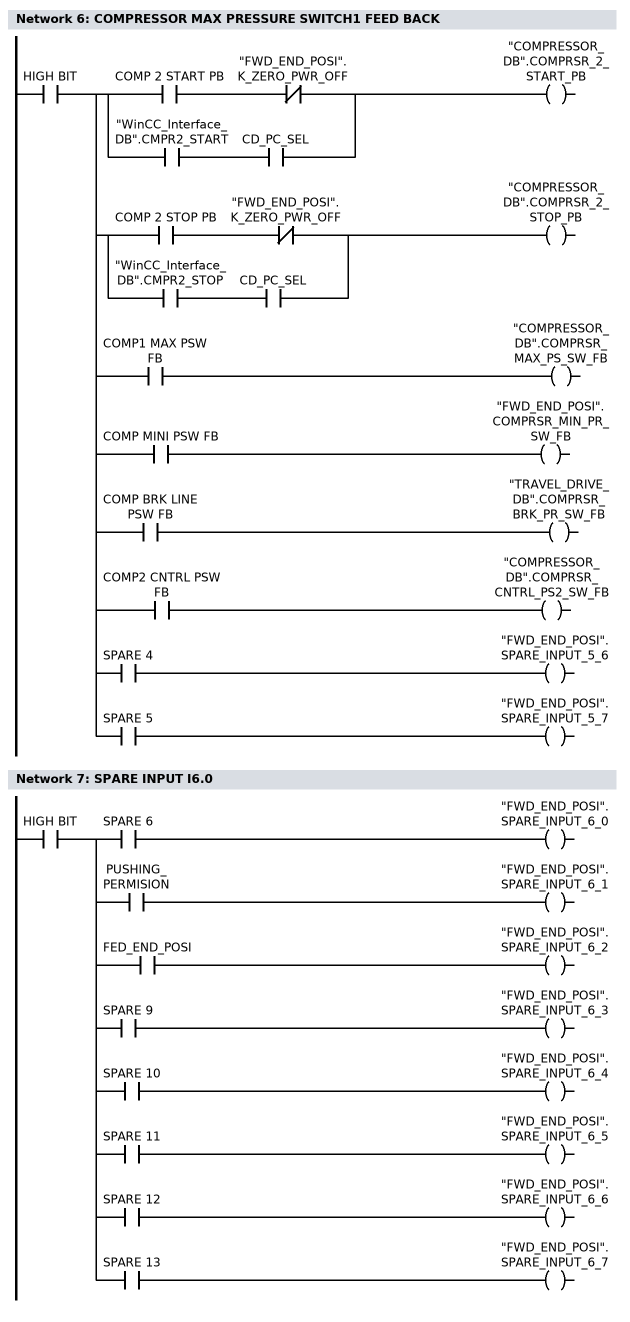
NETWORK
TITLE = COMPRESSOR MAX PRESSURE SWITCH1 FEED BACK
      A     "HIGH BIT";
      =     L 0.0;
      A     L 0.0;
      A(;
      A     "COMP 2 START PB";
      AN    "FWD_END_POSI".K_ZERO_PWR_OFF;
      O;
      A     "WinCC_Interface_DB".CMPR2_START;
      A     "CD_PC_SEL";
      );
      =     "COMPRESSOR_DB".COMPRSR_2_START_PB;
      A     L 0.0;
      A(;
      A     "COMP 2 STOP PB";
      AN    "FWD_END_POSI".K_ZERO_PWR_OFF;
      O;
      A     "WinCC_Interface_DB".CMPR2_STOP;
      A     "CD_PC_SEL";
      );
      =     "COMPRESSOR_DB".COMPRSR_2_STOP_PB;
      A     L 0.0;
      A     "COMP1 MAX PSW FB";
      =     "COMPRESSOR_DB".COMPRSR_MAX_PS_SW_FB;
      A     L 0.0;
      A     "COMP MINI PSW FB";
      =     "FWD_END_POSI".COMPRSR_MIN_PR_SW_FB;
      A     L 0.0;
      A     "COMP BRK LINE PSW FB";
      =     "TRAVEL_DRIVE_DB".COMPRSR_BRK_PR_SW_FB;
      A     L 0.0;
      A     "COMP2 CNTRL PSW FB";
      =     "COMPRESSOR_DB".COMPRSR_CNTRL_PS2_SW_FB;
      A     L 0.0;
      A     "SPARE 4";
      =     "FWD_END_POSI".SPARE_INPUT_5_6;
      A     L 0.0;
      A     "SPARE 5";
      =     "FWD_END_POSI".SPARE_INPUT_5_7;
NETWORK
TITLE = SPARE INPUT I6.0
      A     "HIGH BIT";
      =     L 0.0;
      A     L 0.0;
      A     "SPARE 6";
      =     "FWD_END_POSI".SPARE_INPUT_6_0;
      A     L 0.0;
      A     "PUSHING_PERMISION";
      =     "FWD_END_POSI".SPARE_INPUT_6_1;
      A     L 0.0;
      A     "FED_END_POSI";
      =     "FWD_END_POSI".SPARE_INPUT_6_2;
      A     L 0.0;
      A     "SPARE 9";
      =     "FWD_END_POSI".SPARE_INPUT_6_3;
      A     L 0.0;
      A     "SPARE 10";
      =     "FWD_END_POSI".SPARE_INPUT_6_4;
      A     L 0.0;
      A     "SPARE 11";
      =     "FWD_END_POSI".SPARE_INPUT_6_5;
      A     L 0.0;
      A     "SPARE 12";
      =     "FWD_END_POSI".SPARE_INPUT_6_6;
      A     L 0.0;
      A     "SPARE 13";
      =     "FWD_END_POSI".SPARE_INPUT_6_7;
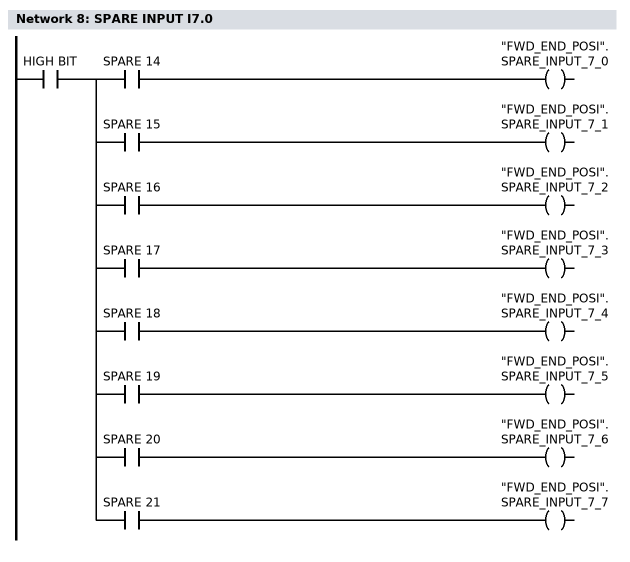
NETWORK
TITLE = SPARE INPUT I7.0
      A     "HIGH BIT";
      =     L 0.0;
      A     L 0.0;
      A     "SPARE 14";
      =     "FWD_END_POSI".SPARE_INPUT_7_0;
      A     L 0.0;
      A     "SPARE 15";
      =     "FWD_END_POSI".SPARE_INPUT_7_1;
      A     L 0.0;
      A     "SPARE 16";
      =     "FWD_END_POSI".SPARE_INPUT_7_2;
      A     L 0.0;
      A     "SPARE 17";
      =     "FWD_END_POSI".SPARE_INPUT_7_3;
      A     L 0.0;
      A     "SPARE 18";
      =     "FWD_END_POSI".SPARE_INPUT_7_4;
      A     L 0.0;
      A     "SPARE 19";
      =     "FWD_END_POSI".SPARE_INPUT_7_5;
      A     L 0.0;
      A     "SPARE 20";
      =     "FWD_END_POSI".SPARE_INPUT_7_6;
      A     L 0.0;
      A     "SPARE 21";
      =     "FWD_END_POSI".SPARE_INPUT_7_7;
END_FUNCTION

FUNCTION "OUTPUT_MAPPING" : VOID	// FC 7
VERSION : 0.1
BEGIN
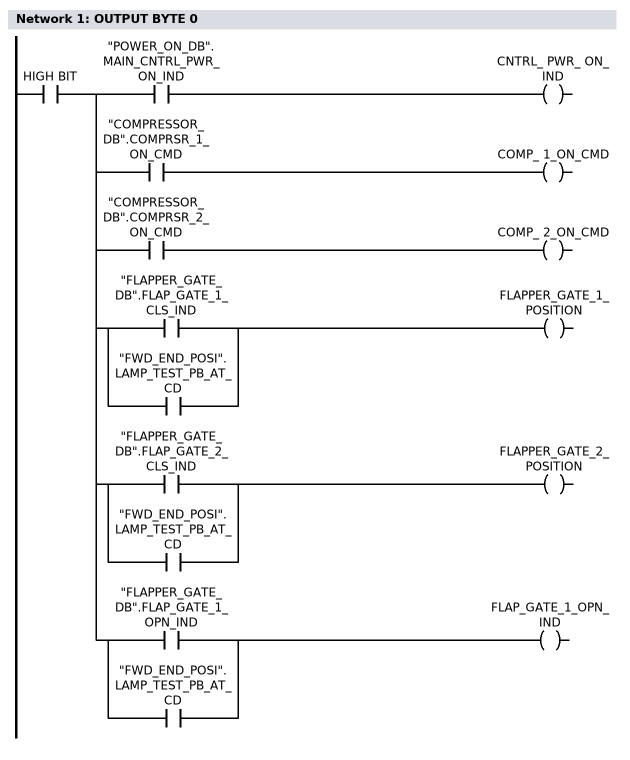
NETWORK
TITLE = OUTPUT BYTE 0
      A     "HIGH BIT";
      =     L 0.0;
      A     L 0.0;
      A     "POWER_ON_DB".MAIN_CNTRL_PWR_ON_IND;
      =     "CNTRL_ PWR_ ON_ IND";
      A     L 0.0;
      A     "COMPRESSOR_DB".COMPRSR_1_ON_CMD;
      =     "COMP_ 1_ON_CMD";
      A     L 0.0;
      A     "COMPRESSOR_DB".COMPRSR_2_ON_CMD;
      =     "COMP_ 2_ON_CMD";
      A     L 0.0;
      A(;
      O     "FLAPPER_GATE_DB".FLAP_GATE_1_CLS_IND;
      O     "FWD_END_POSI".LAMP_TEST_PB_AT_CD;
      );
      =     "FLAPPER_GATE_1_POSITION";
      A     L 0.0;
      A(;
      O     "FLAPPER_GATE_DB".FLAP_GATE_2_CLS_IND;
      O     "FWD_END_POSI".LAMP_TEST_PB_AT_CD;
      );
      =     "FLAPPER_GATE_2_POSITION";
      A     L 0.0;
      A(;
      O     "FLAPPER_GATE_DB".FLAP_GATE_1_OPN_IND;
      O     "FWD_END_POSI".LAMP_TEST_PB_AT_CD;
      );
      =     "FLAP_GATE_1_OPN_IND";
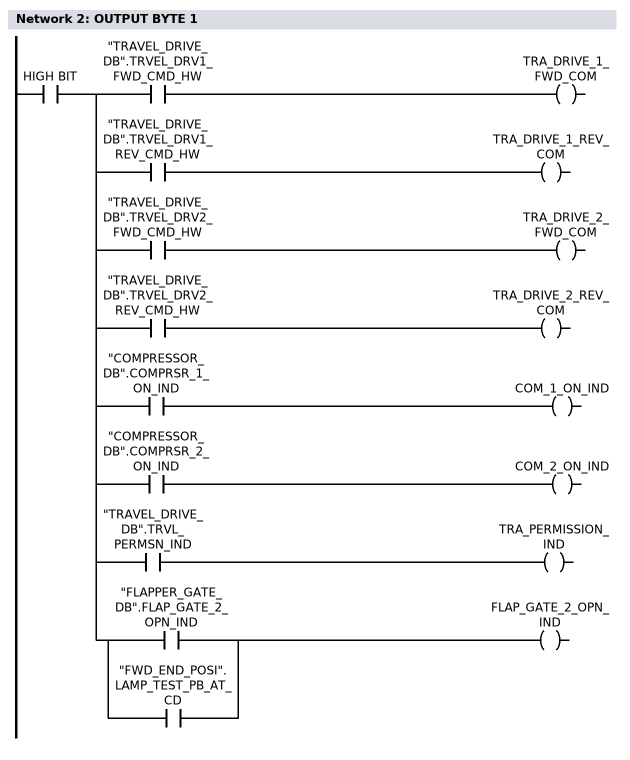
NETWORK
TITLE = OUTPUT BYTE 1
      A     "HIGH BIT";
      =     L 0.0;
      A     L 0.0;
      A     "TRAVEL_DRIVE_DB".TRVEL_DRV1_FWD_CMD_HW;
      =     "TRA_DRIVE_1_FWD_COM";
      A     L 0.0;
      A     "TRAVEL_DRIVE_DB".TRVEL_DRV1_REV_CMD_HW;
      =     "TRA_DRIVE_1_REV_COM";
      A     L 0.0;
      A     "TRAVEL_DRIVE_DB".TRVEL_DRV2_FWD_CMD_HW;
      =     "TRA_DRIVE_2_FWD_COM";
      A     L 0.0;
      A     "TRAVEL_DRIVE_DB".TRVEL_DRV2_REV_CMD_HW;
      =     "TRA_DRIVE_2_REV_COM";
      A     L 0.0;
      A     "COMPRESSOR_DB".COMPRSR_1_ON_IND;
      =     "COM_1_ON_IND";
      A     L 0.0;
      A     "COMPRESSOR_DB".COMPRSR_2_ON_IND;
      =     "COM_2_ON_IND";
      A     L 0.0;
      A     "TRAVEL_DRIVE_DB".TRVL_PERMSN_IND;
      =     "TRA_PERMISSION_IND";
      A     L 0.0;
      A(;
      O     "FLAPPER_GATE_DB".FLAP_GATE_2_OPN_IND;
      O     "FWD_END_POSI".LAMP_TEST_PB_AT_CD;
      );
      =     "FLAP_GATE_2_OPN_IND";
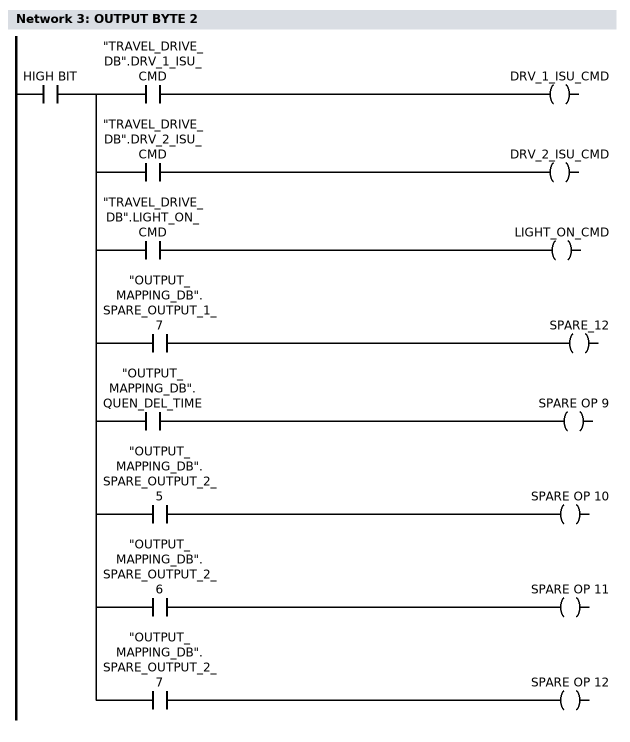
NETWORK
TITLE = OUTPUT BYTE 2
      A     "HIGH BIT";
      =     L 0.0;
      A     L 0.0;
      A     "TRAVEL_DRIVE_DB".DRV_1_ISU_CMD;
      =     "DRV_1_ISU_CMD";
      A     L 0.0;
      A     "TRAVEL_DRIVE_DB".DRV_2_ISU_CMD;
      =     "DRV_2_ISU_CMD";
      A     L 0.0;
      A     "TRAVEL_DRIVE_DB".LIGHT_ON_CMD;
      =     "LIGHT_ON_CMD";
      A     L 0.0;
      A     "OUTPUT_MAPPING_DB".SPARE_OUTPUT_1_7;
      =     "SPARE_12";
      A     L 0.0;
      A     "OUTPUT_MAPPING_DB".QUEN_DEL_TIME;
      =     "SPARE OP 9";
      A     L 0.0;
      A     "OUTPUT_MAPPING_DB".SPARE_OUTPUT_2_5;
      =     "SPARE OP 10";
      A     L 0.0;
      A     "OUTPUT_MAPPING_DB".SPARE_OUTPUT_2_6;
      =     "SPARE OP 11";
      A     L 0.0;
      A     "OUTPUT_MAPPING_DB".SPARE_OUTPUT_2_7;
      =     "SPARE OP 12";
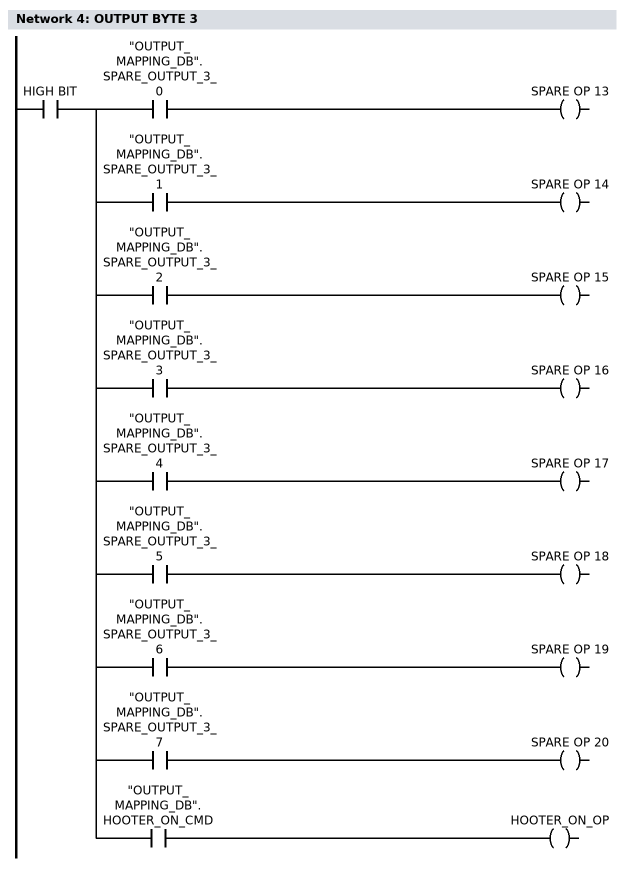
NETWORK
TITLE = OUTPUT BYTE 3
      A     "HIGH BIT";
      =     L 0.0;
      A     L 0.0;
      A     "OUTPUT_MAPPING_DB".SPARE_OUTPUT_3_0;
      =     "SPARE OP 13";
      A     L 0.0;
      A     "OUTPUT_MAPPING_DB".SPARE_OUTPUT_3_1;
      =     "SPARE OP 14";
      A     L 0.0;
      A     "OUTPUT_MAPPING_DB".SPARE_OUTPUT_3_2;
      =     "SPARE OP 15";
      A     L 0.0;
      A     "OUTPUT_MAPPING_DB".SPARE_OUTPUT_3_3;
      =     "SPARE OP 16";
      A     L 0.0;
      A     "OUTPUT_MAPPING_DB".SPARE_OUTPUT_3_4;
      =     "SPARE OP 17";
      A     L 0.0;
      A     "OUTPUT_MAPPING_DB".SPARE_OUTPUT_3_5;
      =     "SPARE OP 18";
      A     L 0.0;
      A     "OUTPUT_MAPPING_DB".SPARE_OUTPUT_3_6;
      =     "SPARE OP 19";
      A     L 0.0;
      A     "OUTPUT_MAPPING_DB".SPARE_OUTPUT_3_7;
      =     "SPARE OP 20";
      A     L 0.0;
      A     "OUTPUT_MAPPING_DB".HOOTER_ON_CMD;
      =     "HOOTER_ON_OP";
END_FUNCTION

FUNCTION "TRAVEL_DRIVE" : VOID	// FC 9
VERSION : 0.1
VAR_TEMP
  TEMP0 : WORD ;
  TEMP1 : WORD ;
  TEMP2 : WORD ;
END_VAR
BEGIN
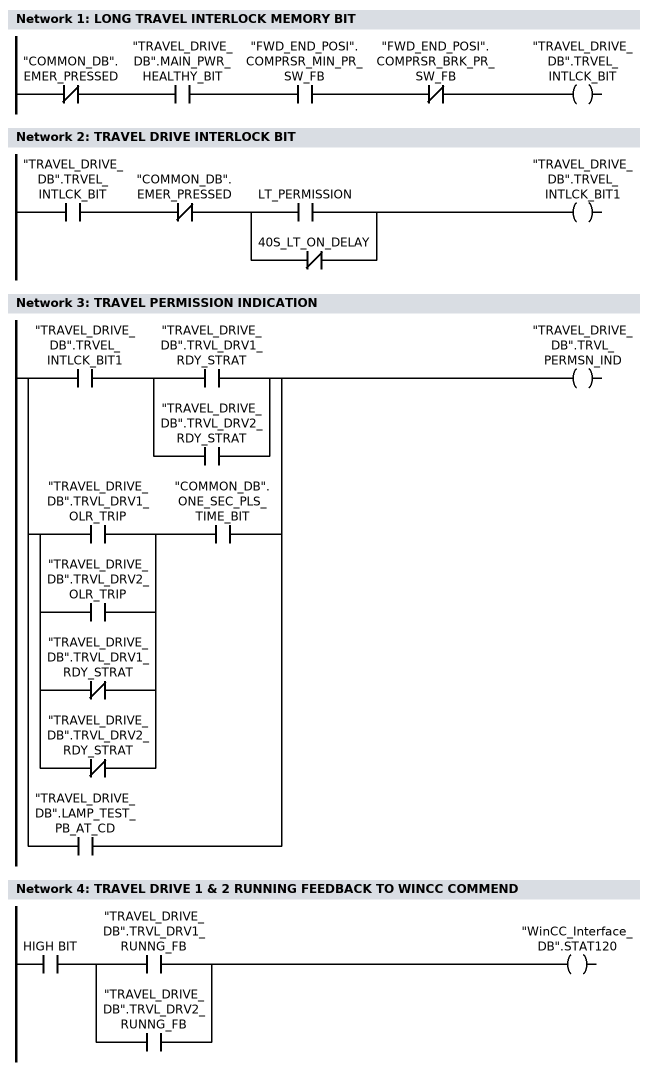
NETWORK
TITLE = LONG TRAVEL INTERLOCK MEMORY BIT
      AN    "COMMON_DB".EMER_PRESSED;
      A     "TRAVEL_DRIVE_DB".MAIN_PWR_HEALTHY_BIT;
      A     "FWD_END_POSI".COMPRSR_MIN_PR_SW_FB;
      AN    "FWD_END_POSI".COMPRSR_BRK_PR_SW_FB;
      =     "TRAVEL_DRIVE_DB".TRVEL_INTLCK_BIT;
NETWORK
TITLE = TRAVEL DRIVE INTERLOCK BIT
      A     "TRAVEL_DRIVE_DB".TRVEL_INTLCK_BIT;
      AN    "COMMON_DB".EMER_PRESSED;
      A(;
      O     "LT_PERMISSION";
      ON    "40S_LT_ON_DELAY";
      );
      =     "TRAVEL_DRIVE_DB".TRVEL_INTLCK_BIT1;
NETWORK
TITLE = TRAVEL PERMISSION INDICATION
      A     "TRAVEL_DRIVE_DB".TRVEL_INTLCK_BIT1;
      A(;
      O     "TRAVEL_DRIVE_DB".TRVL_DRV1_RDY_STRAT;
      O     "TRAVEL_DRIVE_DB".TRVL_DRV2_RDY_STRAT;
      );
      O;
      A(;
      O     "TRAVEL_DRIVE_DB".TRVL_DRV1_OLR_TRIP;
      O     "TRAVEL_DRIVE_DB".TRVL_DRV2_OLR_TRIP;
      ON    "TRAVEL_DRIVE_DB".TRVL_DRV1_RDY_STRAT;
      ON    "TRAVEL_DRIVE_DB".TRVL_DRV2_RDY_STRAT;
      );
      A     "COMMON_DB".ONE_SEC_PLS_TIME_BIT;
      O     "TRAVEL_DRIVE_DB".LAMP_TEST_PB_AT_CD;
      =     "TRAVEL_DRIVE_DB".TRVL_PERMSN_IND;
NETWORK
TITLE = TRAVEL DRIVE 1 & 2 RUNNING FEEDBACK TO WINCC COMMEND
      A     "HIGH BIT";
      A(;
      O     "TRAVEL_DRIVE_DB".TRVL_DRV1_RUNNG_FB;
      O     "TRAVEL_DRIVE_DB".TRVL_DRV2_RUNNG_FB;
      );
      =     "WinCC_Interface_DB".STAT120;
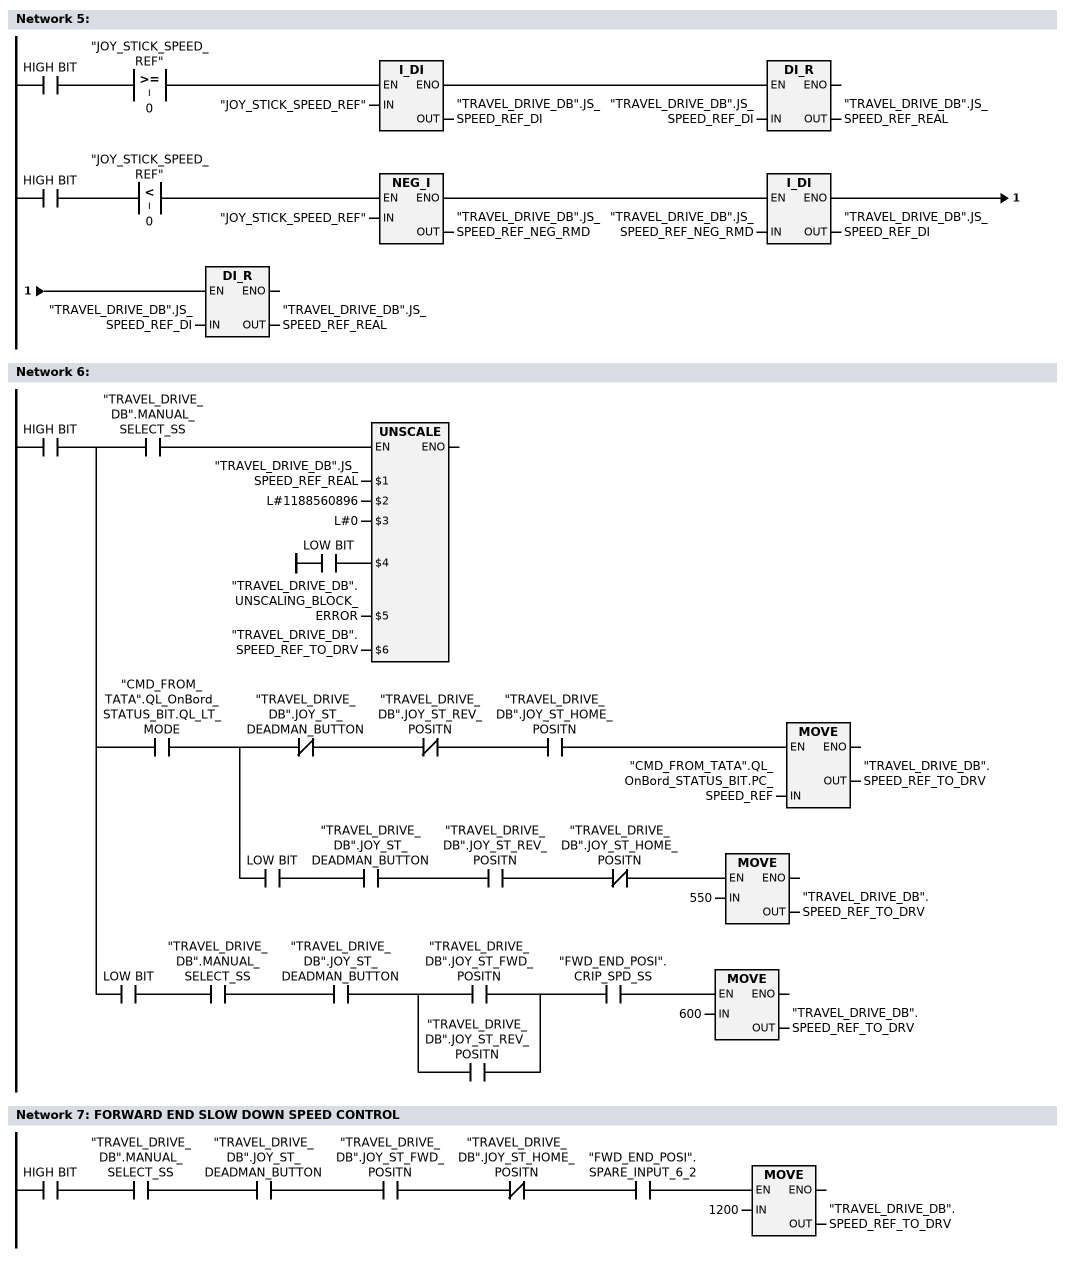
NETWORK
TITLE =
      A     "HIGH BIT";
      =     L 6.0;
      A(;
      A     L 6.0;
      A(;
      L     "JOY_STICK_SPEED_REF";
      L     0;
      >=I;
      );
      JNB   _001;
      L     "JOY_STICK_SPEED_REF";
      ITD;
      T     "TRAVEL_DRIVE_DB".JS_SPEED_REF_DI;
      SET;
      SAVE;
      CLR;
_001: A     BR;
      );
      JNB   _002;
      L     "TRAVEL_DRIVE_DB".JS_SPEED_REF_DI;
      DTR;
      T     "TRAVEL_DRIVE_DB".JS_SPEED_REF_REAL;
_002: NOP   0;
      A(;
      A(;
      A     L 6.0;
      A(;
      L     "JOY_STICK_SPEED_REF";
      L     0;
      <I;
      );
      JNB   _003;
      L     "JOY_STICK_SPEED_REF";
      NEGI;
      T     "TRAVEL_DRIVE_DB".JS_SPEED_REF_NEG_RMD;
      AN    OV;
      SAVE;
      CLR;
_003: A     BR;
      );
      JNB   _004;
      L     "TRAVEL_DRIVE_DB".JS_SPEED_REF_NEG_RMD;
      ITD;
      T     "TRAVEL_DRIVE_DB".JS_SPEED_REF_DI;
      SET;
      SAVE;
      CLR;
_004: A     BR;
      );
      JNB   _005;
      L     "TRAVEL_DRIVE_DB".JS_SPEED_REF_DI;
      DTR;
      T     "TRAVEL_DRIVE_DB".JS_SPEED_REF_REAL;
_005: NOP   0;
NETWORK
TITLE =
      A     "HIGH BIT";
      =     L 6.0;
      A     "LOW BIT";
      =     L 6.1;
      BLD   103;
      A     L 6.0;
      A     "TRAVEL_DRIVE_DB".MANUAL_SELECT_SS;
      JNB   _006;
      CALL  "UNSCALE" (
           $1                       := "TRAVEL_DRIVE_DB".JS_SPEED_REF_REAL,
           $2                       := L#1188560896,
           $3                       := L#0,
           $4                       := L 6.1,
           $5                       := "TRAVEL_DRIVE_DB".UNSCALING_BLOCK_ERROR,
           $6                       := "TRAVEL_DRIVE_DB".SPEED_REF_TO_DRV);
_006: NOP   0;
      A     L 6.0;
      A     "CMD_FROM_TATA".QL_OnBord_STATUS_BIT.QL_LT_MODE;
      =     L 6.1;
      A     L 6.1;
      AN    "TRAVEL_DRIVE_DB".JOY_ST_DEADMAN_BUTTON;
      AN    "TRAVEL_DRIVE_DB".JOY_ST_REV_POSITN;
      A     "TRAVEL_DRIVE_DB".JOY_ST_HOME_POSITN;
      JNB   _007;
      L     "CMD_FROM_TATA".QL_OnBord_STATUS_BIT.PC_SPEED_REF;
      T     "TRAVEL_DRIVE_DB".SPEED_REF_TO_DRV;
_007: NOP   0;
      A     L 6.1;
      A     "LOW BIT";
      A     "TRAVEL_DRIVE_DB".JOY_ST_DEADMAN_BUTTON;
      A     "TRAVEL_DRIVE_DB".JOY_ST_REV_POSITN;
      AN    "TRAVEL_DRIVE_DB".JOY_ST_HOME_POSITN;
      JNB   _008;
      L     550;
      T     "TRAVEL_DRIVE_DB".SPEED_REF_TO_DRV;
_008: NOP   0;
      A     L 6.0;
      A     "LOW BIT";
      A     "TRAVEL_DRIVE_DB".MANUAL_SELECT_SS;
      A     "TRAVEL_DRIVE_DB".JOY_ST_DEADMAN_BUTTON;
      A(;
      O     "TRAVEL_DRIVE_DB".JOY_ST_FWD_POSITN;
      O     "TRAVEL_DRIVE_DB".JOY_ST_REV_POSITN;
      );
      A     "FWD_END_POSI".CRIP_SPD_SS;
      JNB   _009;
      L     600;
      T     "TRAVEL_DRIVE_DB".SPEED_REF_TO_DRV;
_009: NOP   0;
NETWORK
TITLE = FORWARD END SLOW DOWN SPEED CONTROL
      A     "HIGH BIT";
      A     "TRAVEL_DRIVE_DB".MANUAL_SELECT_SS;
      A     "TRAVEL_DRIVE_DB".JOY_ST_DEADMAN_BUTTON;
      A     "TRAVEL_DRIVE_DB".JOY_ST_FWD_POSITN;
      AN    "TRAVEL_DRIVE_DB".JOY_ST_HOME_POSITN;
      A     "FWD_END_POSI".SPARE_INPUT_6_2;
      JNB   _00a;
      L     1200;
      T     "TRAVEL_DRIVE_DB".SPEED_REF_TO_DRV;
_00a: NOP   0;
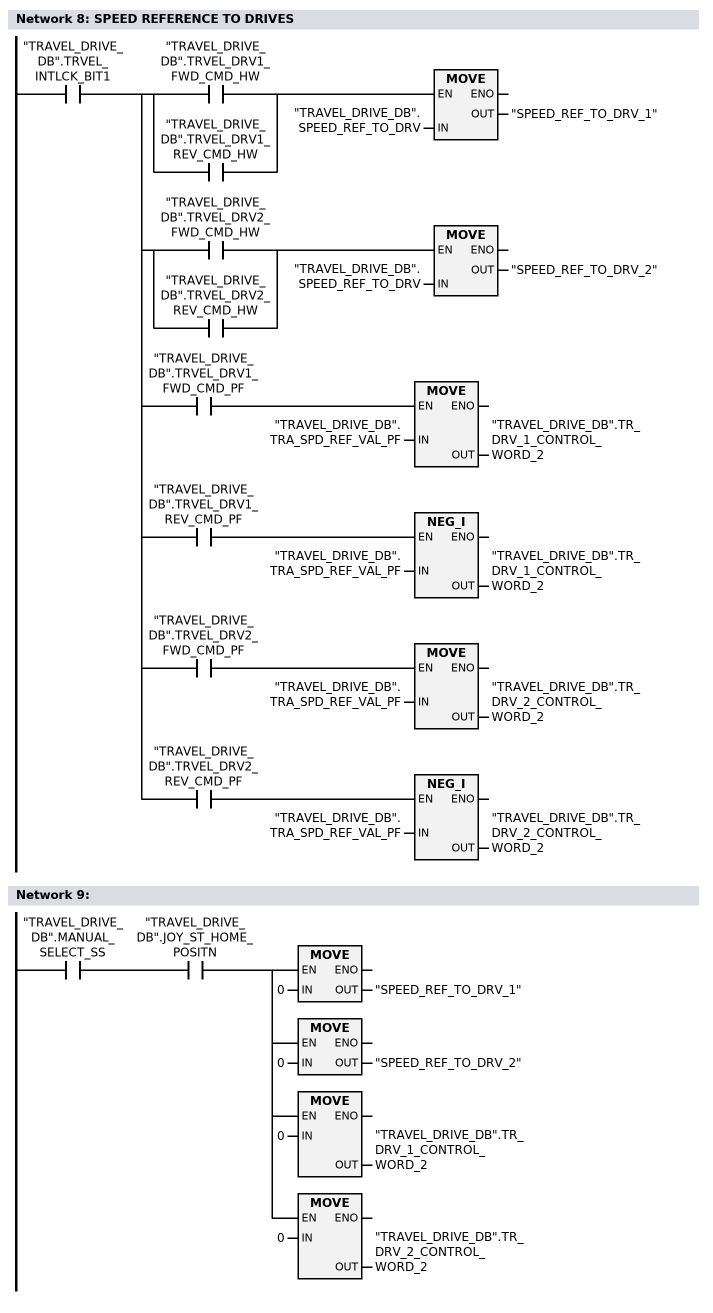
NETWORK
TITLE = SPEED REFERENCE TO DRIVES
      A     "TRAVEL_DRIVE_DB".TRVEL_INTLCK_BIT1;
      =     L 6.0;
      A     L 6.0;
      A(;
      O     "TRAVEL_DRIVE_DB".TRVEL_DRV1_FWD_CMD_HW;
      O     "TRAVEL_DRIVE_DB".TRVEL_DRV1_REV_CMD_HW;
      );
      JNB   _00b;
      L     "TRAVEL_DRIVE_DB".SPEED_REF_TO_DRV;
      T     "SPEED_REF_TO_DRV_1";
_00b: NOP   0;
      A     L 6.0;
      A(;
      O     "TRAVEL_DRIVE_DB".TRVEL_DRV2_FWD_CMD_HW;
      O     "TRAVEL_DRIVE_DB".TRVEL_DRV2_REV_CMD_HW;
      );
      JNB   _00c;
      L     "TRAVEL_DRIVE_DB".SPEED_REF_TO_DRV;
      T     "SPEED_REF_TO_DRV_2";
_00c: NOP   0;
      A     L 6.0;
      A     "TRAVEL_DRIVE_DB".TRVEL_DRV1_FWD_CMD_PF;
      JNB   _00d;
      L     "TRAVEL_DRIVE_DB".TRA_SPD_REF_VAL_PF;
      T     "TRAVEL_DRIVE_DB".TR_DRV_1_CONTROL_WORD_2;
_00d: NOP   0;
      A     L 6.0;
      A     "TRAVEL_DRIVE_DB".TRVEL_DRV1_REV_CMD_PF;
      JNB   _00e;
      L     "TRAVEL_DRIVE_DB".TRA_SPD_REF_VAL_PF;
      NEGI;
      T     "TRAVEL_DRIVE_DB".TR_DRV_1_CONTROL_WORD_2;
_00e: NOP   0;
      A     L 6.0;
      A     "TRAVEL_DRIVE_DB".TRVEL_DRV2_FWD_CMD_PF;
      JNB   _00f;
      L     "TRAVEL_DRIVE_DB".TRA_SPD_REF_VAL_PF;
      T     "TRAVEL_DRIVE_DB".TR_DRV_2_CONTROL_WORD_2;
_00f: NOP   0;
      A     L 6.0;
      A     "TRAVEL_DRIVE_DB".TRVEL_DRV2_REV_CMD_PF;
      JNB   _010;
      L     "TRAVEL_DRIVE_DB".TRA_SPD_REF_VAL_PF;
      NEGI;
      T     "TRAVEL_DRIVE_DB".TR_DRV_2_CONTROL_WORD_2;
_010: NOP   0;
NETWORK
TITLE =
      A     "TRAVEL_DRIVE_DB".MANUAL_SELECT_SS;
      A     "TRAVEL_DRIVE_DB".JOY_ST_HOME_POSITN;
      =     L 6.0;
      A     L 6.0;
      JNB   _011;
      L     0;
      T     "SPEED_REF_TO_DRV_1";
_011: NOP   0;
      A     L 6.0;
      JNB   _012;
      L     0;
      T     "SPEED_REF_TO_DRV_2";
_012: NOP   0;
      A     L 6.0;
      JNB   _013;
      L     0;
      T     "TRAVEL_DRIVE_DB".TR_DRV_1_CONTROL_WORD_2;
_013: NOP   0;
      A     L 6.0;
      JNB   _014;
      L     0;
      T     "TRAVEL_DRIVE_DB".TR_DRV_2_CONTROL_WORD_2;
_014: NOP   0;
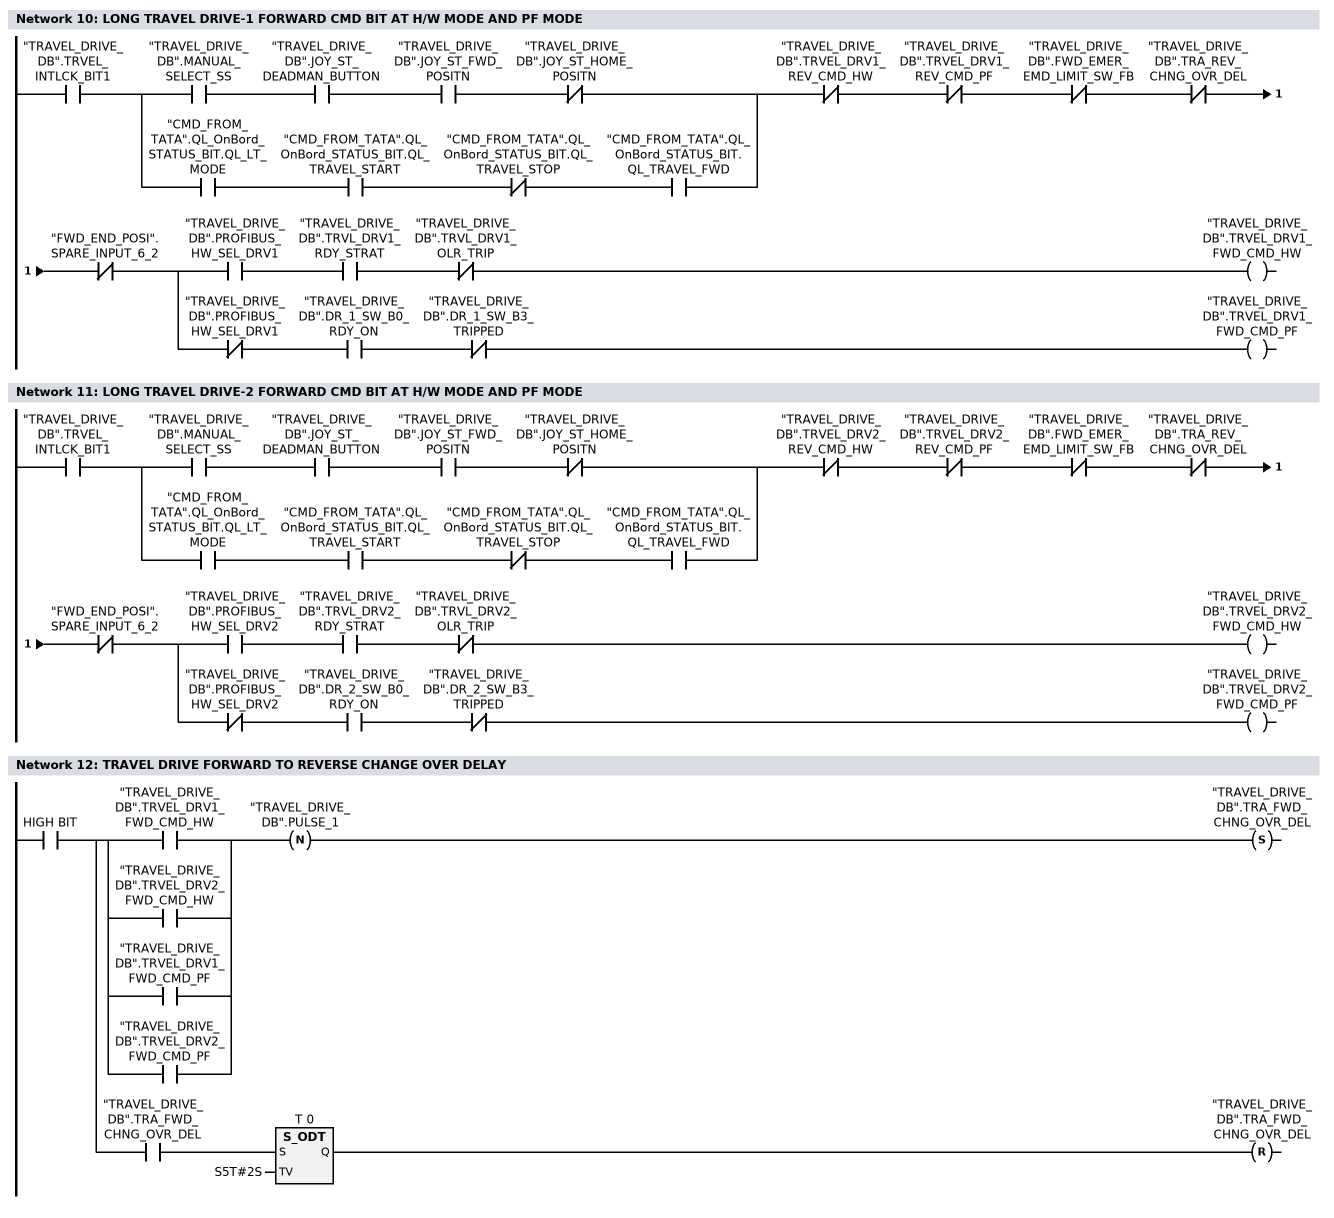
NETWORK
TITLE = LONG TRAVEL DRIVE-1 FORWARD CMD BIT AT H/W MODE AND PF MODE
      A     "TRAVEL_DRIVE_DB".TRVEL_INTLCK_BIT1;
      A(;
      A     "TRAVEL_DRIVE_DB".MANUAL_SELECT_SS;
      A     "TRAVEL_DRIVE_DB".JOY_ST_DEADMAN_BUTTON;
      A     "TRAVEL_DRIVE_DB".JOY_ST_FWD_POSITN;
      AN    "TRAVEL_DRIVE_DB".JOY_ST_HOME_POSITN;
      O;
      A     "CMD_FROM_TATA".QL_OnBord_STATUS_BIT.QL_LT_MODE;
      A     "CMD_FROM_TATA".QL_OnBord_STATUS_BIT.QL_TRAVEL_START;
      AN    "CMD_FROM_TATA".QL_OnBord_STATUS_BIT.QL_TRAVEL_STOP;
      A     "CMD_FROM_TATA".QL_OnBord_STATUS_BIT.QL_TRAVEL_FWD;
      );
      AN    "TRAVEL_DRIVE_DB".TRVEL_DRV1_REV_CMD_HW;
      AN    "TRAVEL_DRIVE_DB".TRVEL_DRV1_REV_CMD_PF;
      AN    "TRAVEL_DRIVE_DB".FWD_EMER_EMD_LIMIT_SW_FB;
      AN    "TRAVEL_DRIVE_DB".TRA_REV_CHNG_OVR_DEL;
      AN    "FWD_END_POSI".SPARE_INPUT_6_2;
      =     L 6.0;
      A     L 6.0;
      A     "TRAVEL_DRIVE_DB".PROFIBUS_HW_SEL_DRV1;
      A     "TRAVEL_DRIVE_DB".TRVL_DRV1_RDY_STRAT;
      AN    "TRAVEL_DRIVE_DB".TRVL_DRV1_OLR_TRIP;
      =     "TRAVEL_DRIVE_DB".TRVEL_DRV1_FWD_CMD_HW;
      A     L 6.0;
      AN    "TRAVEL_DRIVE_DB".PROFIBUS_HW_SEL_DRV1;
      A     "TRAVEL_DRIVE_DB".DR_1_SW_B0_RDY_ON;
      AN    "TRAVEL_DRIVE_DB".DR_1_SW_B3_TRIPPED;
      =     "TRAVEL_DRIVE_DB".TRVEL_DRV1_FWD_CMD_PF;
NETWORK
TITLE = LONG TRAVEL DRIVE-2 FORWARD CMD BIT AT H/W MODE AND PF MODE
      A     "TRAVEL_DRIVE_DB".TRVEL_INTLCK_BIT1;
      A(;
      A     "TRAVEL_DRIVE_DB".MANUAL_SELECT_SS;
      A     "TRAVEL_DRIVE_DB".JOY_ST_DEADMAN_BUTTON;
      A     "TRAVEL_DRIVE_DB".JOY_ST_FWD_POSITN;
      AN    "TRAVEL_DRIVE_DB".JOY_ST_HOME_POSITN;
      O;
      A     "CMD_FROM_TATA".QL_OnBord_STATUS_BIT.QL_LT_MODE;
      A     "CMD_FROM_TATA".QL_OnBord_STATUS_BIT.QL_TRAVEL_START;
      AN    "CMD_FROM_TATA".QL_OnBord_STATUS_BIT.QL_TRAVEL_STOP;
      A     "CMD_FROM_TATA".QL_OnBord_STATUS_BIT.QL_TRAVEL_FWD;
      );
      AN    "TRAVEL_DRIVE_DB".TRVEL_DRV2_REV_CMD_HW;
      AN    "TRAVEL_DRIVE_DB".TRVEL_DRV2_REV_CMD_PF;
      AN    "TRAVEL_DRIVE_DB".FWD_EMER_EMD_LIMIT_SW_FB;
      AN    "TRAVEL_DRIVE_DB".TRA_REV_CHNG_OVR_DEL;
      AN    "FWD_END_POSI".SPARE_INPUT_6_2;
      =     L 6.0;
      A     L 6.0;
      A     "TRAVEL_DRIVE_DB".PROFIBUS_HW_SEL_DRV2;
      A     "TRAVEL_DRIVE_DB".TRVL_DRV2_RDY_STRAT;
      AN    "TRAVEL_DRIVE_DB".TRVL_DRV2_OLR_TRIP;
      =     "TRAVEL_DRIVE_DB".TRVEL_DRV2_FWD_CMD_HW;
      A     L 6.0;
      AN    "TRAVEL_DRIVE_DB".PROFIBUS_HW_SEL_DRV2;
      A     "TRAVEL_DRIVE_DB".DR_2_SW_B0_RDY_ON;
      AN    "TRAVEL_DRIVE_DB".DR_2_SW_B3_TRIPPED;
      =     "TRAVEL_DRIVE_DB".TRVEL_DRV2_FWD_CMD_PF;
NETWORK
TITLE = TRAVEL DRIVE FORWARD TO REVERSE CHANGE OVER DELAY
      A     "HIGH BIT";
      =     L 6.0;
      A     L 6.0;
      A(;
      O     "TRAVEL_DRIVE_DB".TRVEL_DRV1_FWD_CMD_HW;
      O     "TRAVEL_DRIVE_DB".TRVEL_DRV2_FWD_CMD_HW;
      O     "TRAVEL_DRIVE_DB".TRVEL_DRV1_FWD_CMD_PF;
      O     "TRAVEL_DRIVE_DB".TRVEL_DRV2_FWD_CMD_PF;
      );
      FN    "TRAVEL_DRIVE_DB".PULSE_1;
      S     "TRAVEL_DRIVE_DB".TRA_FWD_CHNG_OVR_DEL;
      A     L 6.0;
      A     "TRAVEL_DRIVE_DB".TRA_FWD_CHNG_OVR_DEL;
      L     S5T#2S;
      SD    T 0;
      NOP   0;
      NOP   0;
      NOP   0;
      A     T 0;
      R     "TRAVEL_DRIVE_DB".TRA_FWD_CHNG_OVR_DEL;
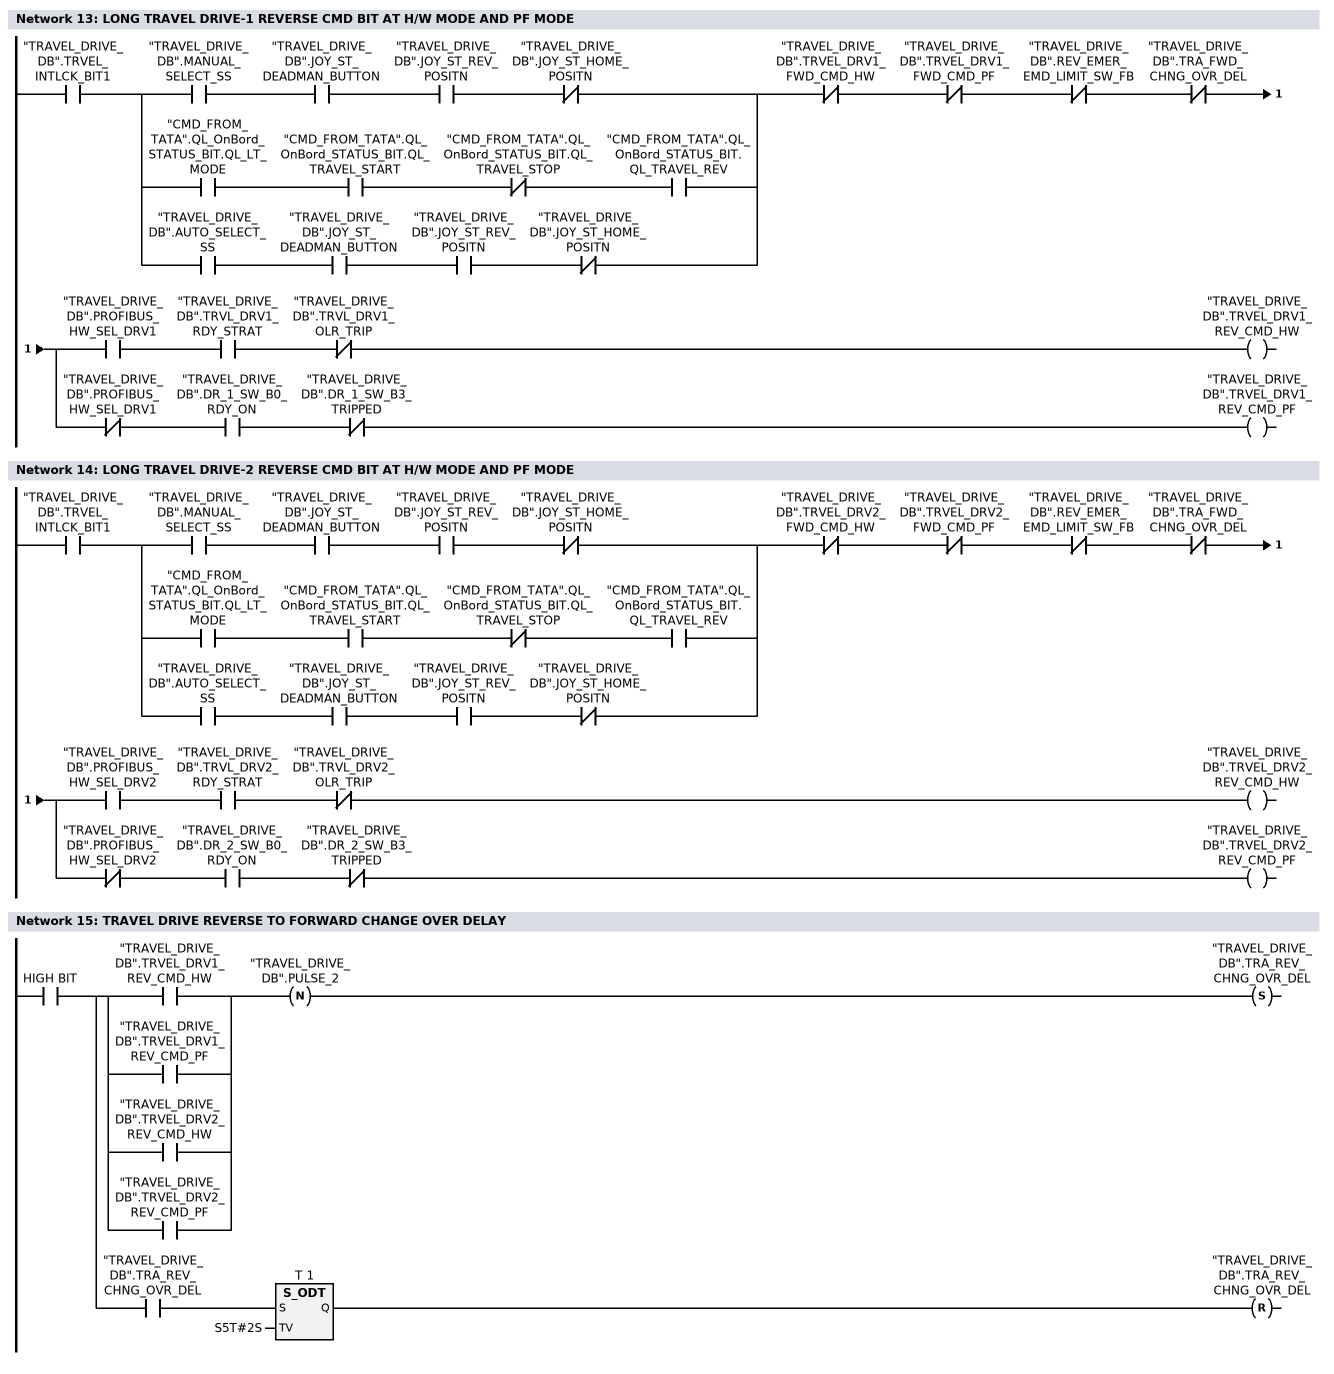
NETWORK
TITLE = LONG TRAVEL DRIVE-1 REVERSE CMD BIT AT H/W MODE AND PF MODE
      A     "TRAVEL_DRIVE_DB".TRVEL_INTLCK_BIT1;
      A(;
      A     "TRAVEL_DRIVE_DB".MANUAL_SELECT_SS;
      A     "TRAVEL_DRIVE_DB".JOY_ST_DEADMAN_BUTTON;
      A     "TRAVEL_DRIVE_DB".JOY_ST_REV_POSITN;
      AN    "TRAVEL_DRIVE_DB".JOY_ST_HOME_POSITN;
      O;
      A     "CMD_FROM_TATA".QL_OnBord_STATUS_BIT.QL_LT_MODE;
      A     "CMD_FROM_TATA".QL_OnBord_STATUS_BIT.QL_TRAVEL_START;
      AN    "CMD_FROM_TATA".QL_OnBord_STATUS_BIT.QL_TRAVEL_STOP;
      A     "CMD_FROM_TATA".QL_OnBord_STATUS_BIT.QL_TRAVEL_REV;
      O;
      A     "TRAVEL_DRIVE_DB".AUTO_SELECT_SS;
      A     "TRAVEL_DRIVE_DB".JOY_ST_DEADMAN_BUTTON;
      A     "TRAVEL_DRIVE_DB".JOY_ST_REV_POSITN;
      AN    "TRAVEL_DRIVE_DB".JOY_ST_HOME_POSITN;
      );
      AN    "TRAVEL_DRIVE_DB".TRVEL_DRV1_FWD_CMD_HW;
      AN    "TRAVEL_DRIVE_DB".TRVEL_DRV1_FWD_CMD_PF;
      AN    "TRAVEL_DRIVE_DB".REV_EMER_EMD_LIMIT_SW_FB;
      AN    "TRAVEL_DRIVE_DB".TRA_FWD_CHNG_OVR_DEL;
      =     L 6.0;
      A     L 6.0;
      A     "TRAVEL_DRIVE_DB".PROFIBUS_HW_SEL_DRV1;
      A     "TRAVEL_DRIVE_DB".TRVL_DRV1_RDY_STRAT;
      AN    "TRAVEL_DRIVE_DB".TRVL_DRV1_OLR_TRIP;
      =     "TRAVEL_DRIVE_DB".TRVEL_DRV1_REV_CMD_HW;
      A     L 6.0;
      AN    "TRAVEL_DRIVE_DB".PROFIBUS_HW_SEL_DRV1;
      A     "TRAVEL_DRIVE_DB".DR_1_SW_B0_RDY_ON;
      AN    "TRAVEL_DRIVE_DB".DR_1_SW_B3_TRIPPED;
      =     "TRAVEL_DRIVE_DB".TRVEL_DRV1_REV_CMD_PF;
NETWORK
TITLE = LONG TRAVEL DRIVE-2 REVERSE CMD BIT AT H/W MODE AND PF MODE
      A     "TRAVEL_DRIVE_DB".TRVEL_INTLCK_BIT1;
      A(;
      A     "TRAVEL_DRIVE_DB".MANUAL_SELECT_SS;
      A     "TRAVEL_DRIVE_DB".JOY_ST_DEADMAN_BUTTON;
      A     "TRAVEL_DRIVE_DB".JOY_ST_REV_POSITN;
      AN    "TRAVEL_DRIVE_DB".JOY_ST_HOME_POSITN;
      O;
      A     "CMD_FROM_TATA".QL_OnBord_STATUS_BIT.QL_LT_MODE;
      A     "CMD_FROM_TATA".QL_OnBord_STATUS_BIT.QL_TRAVEL_START;
      AN    "CMD_FROM_TATA".QL_OnBord_STATUS_BIT.QL_TRAVEL_STOP;
      A     "CMD_FROM_TATA".QL_OnBord_STATUS_BIT.QL_TRAVEL_REV;
      O;
      A     "TRAVEL_DRIVE_DB".AUTO_SELECT_SS;
      A     "TRAVEL_DRIVE_DB".JOY_ST_DEADMAN_BUTTON;
      A     "TRAVEL_DRIVE_DB".JOY_ST_REV_POSITN;
      AN    "TRAVEL_DRIVE_DB".JOY_ST_HOME_POSITN;
      );
      AN    "TRAVEL_DRIVE_DB".TRVEL_DRV2_FWD_CMD_HW;
      AN    "TRAVEL_DRIVE_DB".TRVEL_DRV2_FWD_CMD_PF;
      AN    "TRAVEL_DRIVE_DB".REV_EMER_EMD_LIMIT_SW_FB;
      AN    "TRAVEL_DRIVE_DB".TRA_FWD_CHNG_OVR_DEL;
      =     L 6.0;
      A     L 6.0;
      A     "TRAVEL_DRIVE_DB".PROFIBUS_HW_SEL_DRV2;
      A     "TRAVEL_DRIVE_DB".TRVL_DRV2_RDY_STRAT;
      AN    "TRAVEL_DRIVE_DB".TRVL_DRV2_OLR_TRIP;
      =     "TRAVEL_DRIVE_DB".TRVEL_DRV2_REV_CMD_HW;
      A     L 6.0;
      AN    "TRAVEL_DRIVE_DB".PROFIBUS_HW_SEL_DRV2;
      A     "TRAVEL_DRIVE_DB".DR_2_SW_B0_RDY_ON;
      AN    "TRAVEL_DRIVE_DB".DR_2_SW_B3_TRIPPED;
      =     "TRAVEL_DRIVE_DB".TRVEL_DRV2_REV_CMD_PF;
NETWORK
TITLE = TRAVEL DRIVE REVERSE TO FORWARD CHANGE OVER DELAY
      A     "HIGH BIT";
      =     L 6.0;
      A     L 6.0;
      A(;
      O     "TRAVEL_DRIVE_DB".TRVEL_DRV1_REV_CMD_HW;
      O     "TRAVEL_DRIVE_DB".TRVEL_DRV1_REV_CMD_PF;
      O     "TRAVEL_DRIVE_DB".TRVEL_DRV2_REV_CMD_HW;
      O     "TRAVEL_DRIVE_DB".TRVEL_DRV2_REV_CMD_PF;
      );
      FN    "TRAVEL_DRIVE_DB".PULSE_2;
      S     "TRAVEL_DRIVE_DB".TRA_REV_CHNG_OVR_DEL;
      A     L 6.0;
      A     "TRAVEL_DRIVE_DB".TRA_REV_CHNG_OVR_DEL;
      L     S5T#2S;
      SD    T 1;
      NOP   0;
      NOP   0;
      NOP   0;
      A     T 1;
      R     "TRAVEL_DRIVE_DB".TRA_REV_CHNG_OVR_DEL;
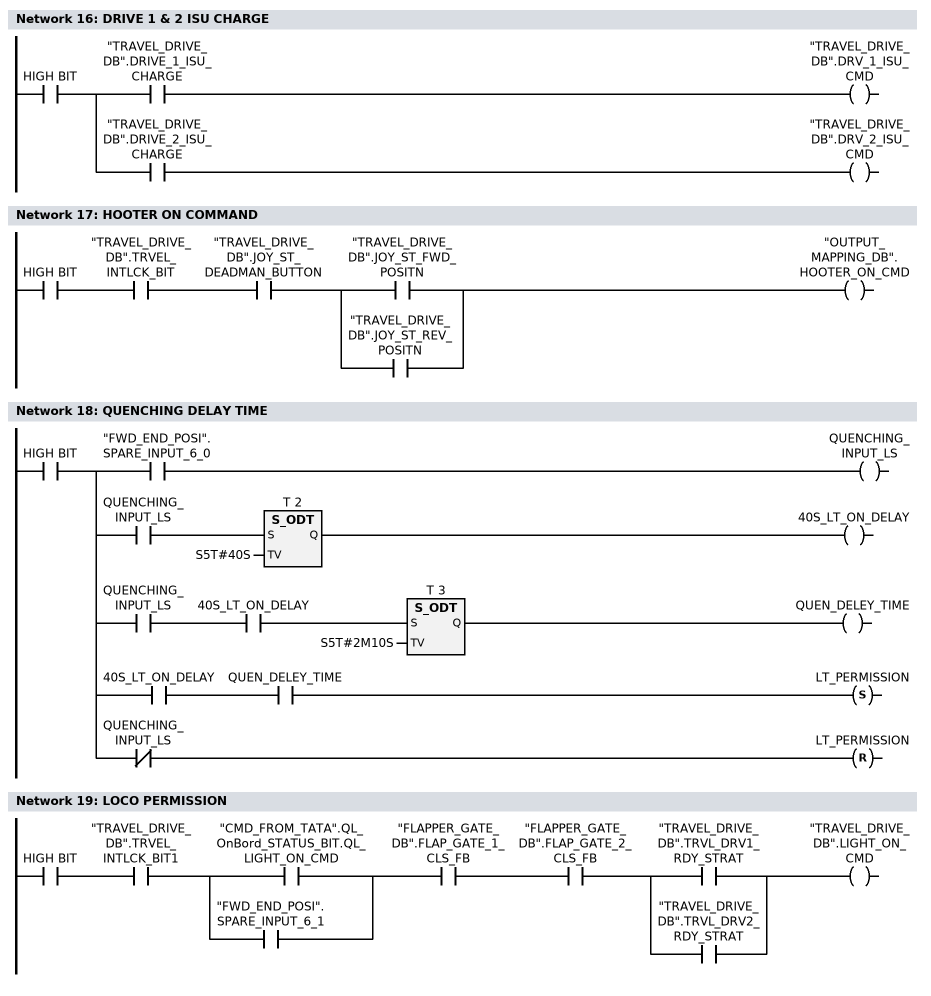
NETWORK
TITLE = DRIVE 1 & 2 ISU CHARGE
      A     "HIGH BIT";
      =     L 6.0;
      A     L 6.0;
      A     "TRAVEL_DRIVE_DB".DRIVE_1_ISU_CHARGE;
      =     "TRAVEL_DRIVE_DB".DRV_1_ISU_CMD;
      A     L 6.0;
      A     "TRAVEL_DRIVE_DB".DRIVE_2_ISU_CHARGE;
      =     "TRAVEL_DRIVE_DB".DRV_2_ISU_CMD;
NETWORK
TITLE = HOOTER ON COMMAND
      A     "HIGH BIT";
      A     "TRAVEL_DRIVE_DB".TRVEL_INTLCK_BIT;
      A     "TRAVEL_DRIVE_DB".JOY_ST_DEADMAN_BUTTON;
      A(;
      O     "TRAVEL_DRIVE_DB".JOY_ST_FWD_POSITN;
      O     "TRAVEL_DRIVE_DB".JOY_ST_REV_POSITN;
      );
      =     "OUTPUT_MAPPING_DB".HOOTER_ON_CMD;
NETWORK
TITLE = QUENCHING DELAY TIME 
      A     "HIGH BIT";
      =     L 6.0;
      A     L 6.0;
      A     "FWD_END_POSI".SPARE_INPUT_6_0;
      =     "QUENCHING_INPUT_LS";
      A     L 6.0;
      A     "QUENCHING_INPUT_LS";
      L     S5T#40S;
      SD    T 2;
      NOP   0;
      NOP   0;
      NOP   0;
      A     T 2;
      =     "40S_LT_ON_DELAY";
      A     L 6.0;
      A     "QUENCHING_INPUT_LS";
      A     "40S_LT_ON_DELAY";
      L     S5T#2M10S;
      SD    T 3;
      NOP   0;
      NOP   0;
      NOP   0;
      A     T 3;
      =     "QUEN_DELEY_TIME";
      A     L 6.0;
      A     "40S_LT_ON_DELAY";
      A     "QUEN_DELEY_TIME";
      S     "LT_PERMISSION";
      A     L 6.0;
      AN    "QUENCHING_INPUT_LS";
      R     "LT_PERMISSION";
NETWORK
TITLE = LOCO PERMISSION
      A     "HIGH BIT";
      A     "TRAVEL_DRIVE_DB".TRVEL_INTLCK_BIT1;
      A(;
      O     "CMD_FROM_TATA".QL_OnBord_STATUS_BIT.QL_LIGHT_ON_CMD;
      O     "FWD_END_POSI".SPARE_INPUT_6_1;
      );
      A     "FLAPPER_GATE_DB".FLAP_GATE_1_CLS_FB;
      A     "FLAPPER_GATE_DB".FLAP_GATE_2_CLS_FB;
      A(;
      O     "TRAVEL_DRIVE_DB".TRVL_DRV1_RDY_STRAT;
      O     "TRAVEL_DRIVE_DB".TRVL_DRV2_RDY_STRAT;
      );
      =     "TRAVEL_DRIVE_DB".LIGHT_ON_CMD;
END_FUNCTION

FUNCTION "PROFIBUS_COMMUNICATION" : VOID	// FC 10
VERSION : 0.1
VAR_TEMP
  TEMP0 : INT ;
  TEMP1 : INT ;
  TEMP2 : INT ;
  TEMP3 : INT ;
  TEMP4 : INT ;
  TEMP5 : INT ;
  TEMP6 : INT ;
  TEMP7 : INT ;
  TEMP8 : INT ;
  TEMP9 : WORD ;
  TEMP10 : WORD ;
END_VAR
BEGIN
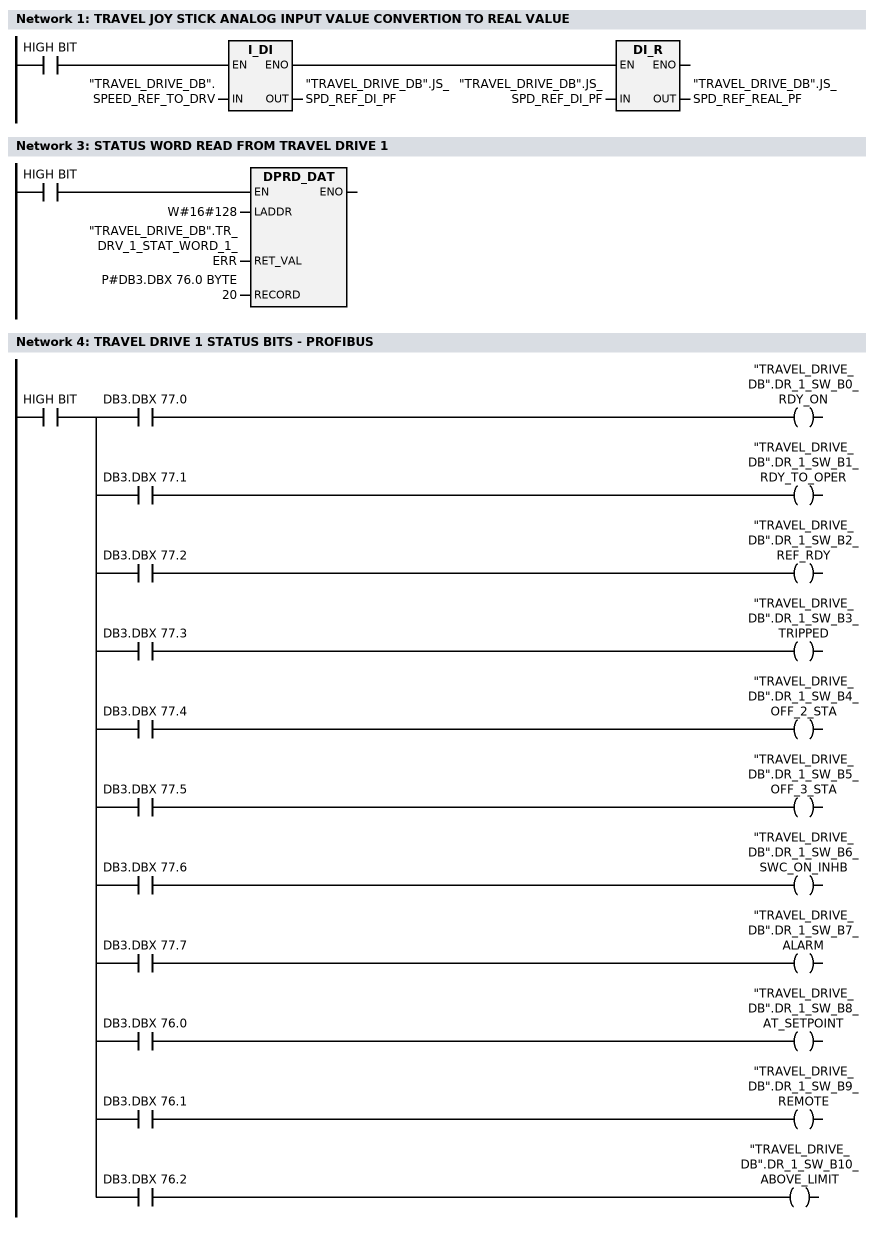
NETWORK
TITLE = TRAVEL JOY STICK ANALOG INPUT VALUE CONVERTION TO REAL VALUE
//TRAVEL DRIVE JOY STICK ANALOG INPUT VALUE CONVERTION TO REAL VALUE
      A(;
      A     "HIGH BIT";
      JNB   _001;
      L     "TRAVEL_DRIVE_DB".SPEED_REF_TO_DRV;
      ITD;
      T     "TRAVEL_DRIVE_DB".JS_SPD_REF_DI_PF;
      SET;
      SAVE;
      CLR;
_001: A     BR;
      );
      JNB   _002;
      L     "TRAVEL_DRIVE_DB".JS_SPD_REF_DI_PF;
      DTR;
      T     "TRAVEL_DRIVE_DB".JS_SPD_REF_REAL_PF;
_002: NOP   0;
NETWORK
TITLE = SCALING FOR PROFIBUS CONTROL SPEED REFERENCE
      A(;
      A(;
      A     "LOW BIT";
      =     L 22.0;
      BLD   103;
      A     "HIGH BIT";
      JNB   _003;
      CALL  "SCALE" (
           $1                       := "TRAVEL_DRIVE_DB".SPEED_REF_TO_DRV,
           $2                       := L#1184645120,
           $3                       := L#0,
           $4                       := L 22.0,
           $5                       := "TRAVEL_DRIVE_DB".JS_SPD_REF_UN_SL_FLT_PF,
           $6                       := "TRAVEL_DRIVE_DB".JS_SPD_REF_REAL_PF);
_003: A     BR;
      );
      JNB   _004;
      L     "TRAVEL_DRIVE_DB".JS_SPD_REF_REAL_PF;
      TRUNC;
      T     "TRAVEL_DRIVE_DB".JS_SPD_REF_DI_PF;
      AN    OV;
      SAVE;
      CLR;
_004: A     BR;
      );
      JNB   _005;
      L     DB3.DBW 242;
      T     "TRAVEL_DRIVE_DB".TRA_SPD_REF_VAL_PF;
_005: NOP   0;
NETWORK
TITLE = STATUS WORD READ FROM TRAVEL DRIVE 1
      A     "HIGH BIT";
      JNB   _006;
      CALL  "DPRD_DAT" (
           LADDR                    := W#16#128,
           RET_VAL                  := "TRAVEL_DRIVE_DB".TR_DRV_1_STAT_WORD_1_ERR,
           RECORD                   := P#DB3.DBX 76.0 BYTE 20);
_006: NOP   0;
NETWORK
TITLE = TRAVEL DRIVE 1 STATUS BITS - PROFIBUS
      A     "HIGH BIT";
      =     L 22.0;
      A     L 22.0;
      A     DB3.DBX 77.0;
      =     "TRAVEL_DRIVE_DB".DR_1_SW_B0_RDY_ON;
      A     L 22.0;
      A     DB3.DBX 77.1;
      =     "TRAVEL_DRIVE_DB".DR_1_SW_B1_RDY_TO_OPER;
      A     L 22.0;
      A     DB3.DBX 77.2;
      =     "TRAVEL_DRIVE_DB".DR_1_SW_B2_REF_RDY;
      A     L 22.0;
      A     DB3.DBX 77.3;
      =     "TRAVEL_DRIVE_DB".DR_1_SW_B3_TRIPPED;
      A     L 22.0;
      A     DB3.DBX 77.4;
      =     "TRAVEL_DRIVE_DB".DR_1_SW_B4_OFF_2_STA;
      A     L 22.0;
      A     DB3.DBX 77.5;
      =     "TRAVEL_DRIVE_DB".DR_1_SW_B5_OFF_3_STA;
      A     L 22.0;
      A     DB3.DBX 77.6;
      =     "TRAVEL_DRIVE_DB".DR_1_SW_B6_SWC_ON_INHB;
      A     L 22.0;
      A     DB3.DBX 77.7;
      =     "TRAVEL_DRIVE_DB".DR_1_SW_B7_ALARM;
      A     L 22.0;
      A     DB3.DBX 76.0;
      =     "TRAVEL_DRIVE_DB".DR_1_SW_B8_AT_SETPOINT;
      A     L 22.0;
      A     DB3.DBX 76.1;
      =     "TRAVEL_DRIVE_DB".DR_1_SW_B9_REMOTE;
      A     L 22.0;
      A     DB3.DBX 76.2;
      =     "TRAVEL_DRIVE_DB".DR_1_SW_B10_ABOVE_LIMIT;
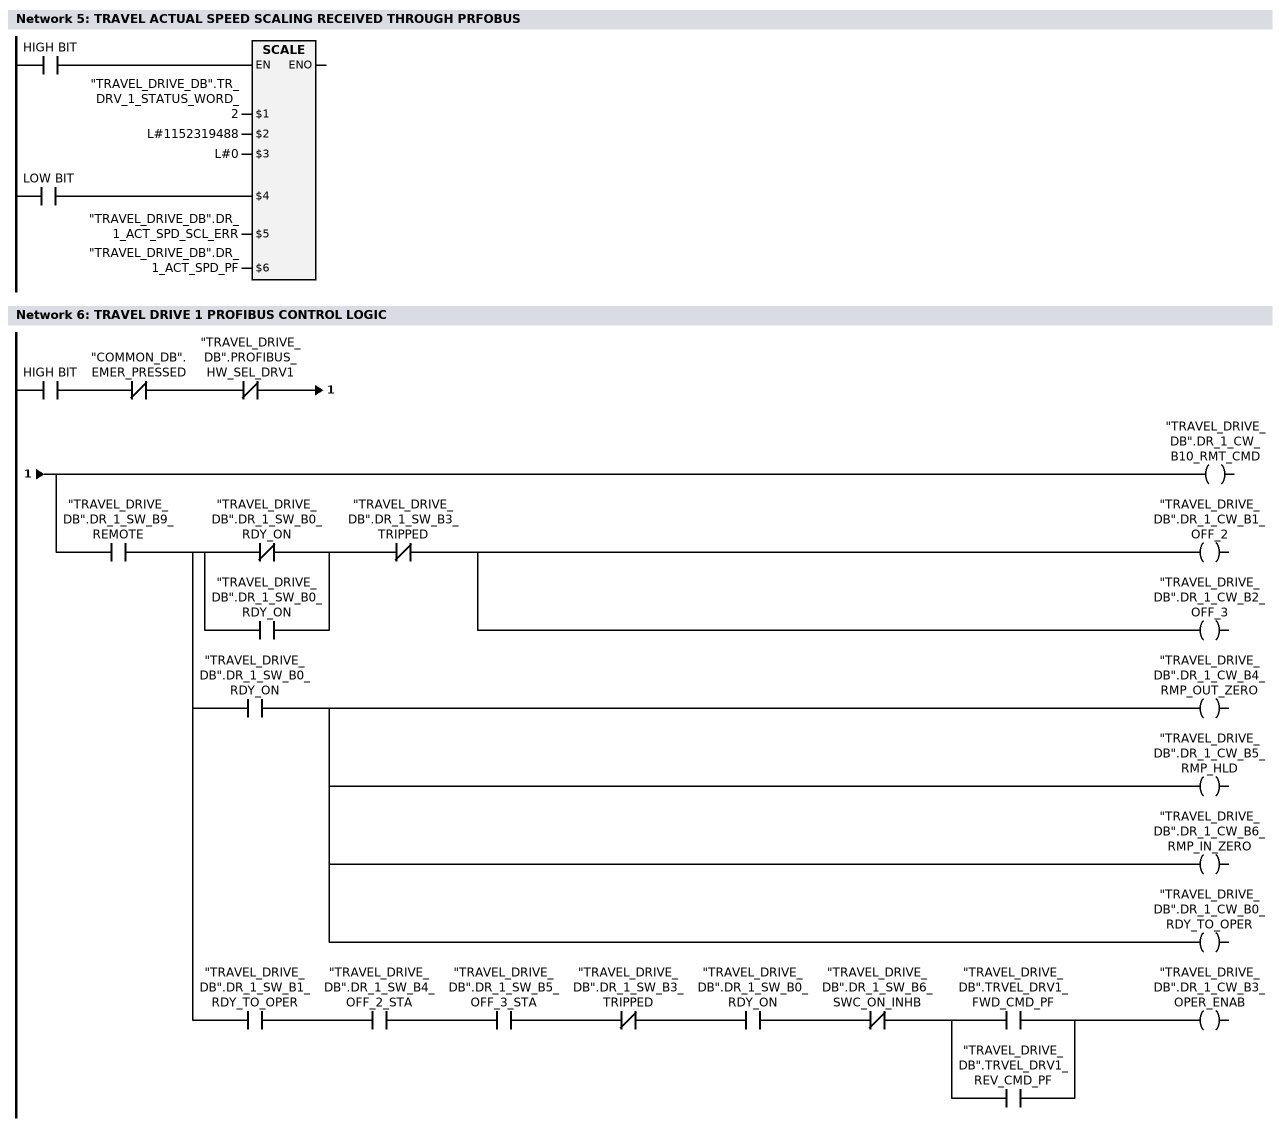
NETWORK
TITLE = TRAVEL ACTUAL SPEED SCALING RECEIVED THROUGH PRFOBUS
      A     "LOW BIT";
      =     L 22.0;
      BLD   103;
      A     "HIGH BIT";
      JNB   _007;
      CALL  "SCALE" (
           $1                       := "TRAVEL_DRIVE_DB".TR_DRV_1_STATUS_WORD_2,
           $2                       := L#1152319488,
           $3                       := L#0,
           $4                       := L 22.0,
           $5                       := "TRAVEL_DRIVE_DB".DR_1_ACT_SPD_SCL_ERR,
           $6                       := "TRAVEL_DRIVE_DB".DR_1_ACT_SPD_PF);
_007: NOP   0;
NETWORK
TITLE = TRAVEL DRIVE 1 PROFIBUS CONTROL LOGIC
      A     "HIGH BIT";
      AN    "COMMON_DB".EMER_PRESSED;
      AN    "TRAVEL_DRIVE_DB".PROFIBUS_HW_SEL_DRV1;
      =     L 22.0;
      A     L 22.0;
      BLD   102;
      =     "TRAVEL_DRIVE_DB".DR_1_CW_B10_RMT_CMD;
      A     L 22.0;
      A     "TRAVEL_DRIVE_DB".DR_1_SW_B9_REMOTE;
      =     L 22.1;
      A     L 22.1;
      A(;
      ON    "TRAVEL_DRIVE_DB".DR_1_SW_B0_RDY_ON;
      O     "TRAVEL_DRIVE_DB".DR_1_SW_B0_RDY_ON;
      );
      AN    "TRAVEL_DRIVE_DB".DR_1_SW_B3_TRIPPED;
      =     "TRAVEL_DRIVE_DB".DR_1_CW_B1_OFF_2;
      =     "TRAVEL_DRIVE_DB".DR_1_CW_B2_OFF_3;
      A     L 22.1;
      A     "TRAVEL_DRIVE_DB".DR_1_SW_B0_RDY_ON;
      =     "TRAVEL_DRIVE_DB".DR_1_CW_B4_RMP_OUT_ZERO;
      =     "TRAVEL_DRIVE_DB".DR_1_CW_B5_RMP_HLD;
      =     "TRAVEL_DRIVE_DB".DR_1_CW_B6_RMP_IN_ZERO;
      =     "TRAVEL_DRIVE_DB".DR_1_CW_B0_RDY_TO_OPER;
      A     L 22.1;
      A     "TRAVEL_DRIVE_DB".DR_1_SW_B1_RDY_TO_OPER;
      A     "TRAVEL_DRIVE_DB".DR_1_SW_B4_OFF_2_STA;
      A     "TRAVEL_DRIVE_DB".DR_1_SW_B5_OFF_3_STA;
      AN    "TRAVEL_DRIVE_DB".DR_1_SW_B3_TRIPPED;
      A     "TRAVEL_DRIVE_DB".DR_1_SW_B0_RDY_ON;
      AN    "TRAVEL_DRIVE_DB".DR_1_SW_B6_SWC_ON_INHB;
      A(;
      O     "TRAVEL_DRIVE_DB".TRVEL_DRV1_FWD_CMD_PF;
      O     "TRAVEL_DRIVE_DB".TRVEL_DRV1_REV_CMD_PF;
      );
      =     "TRAVEL_DRIVE_DB".DR_1_CW_B3_OPER_ENAB;
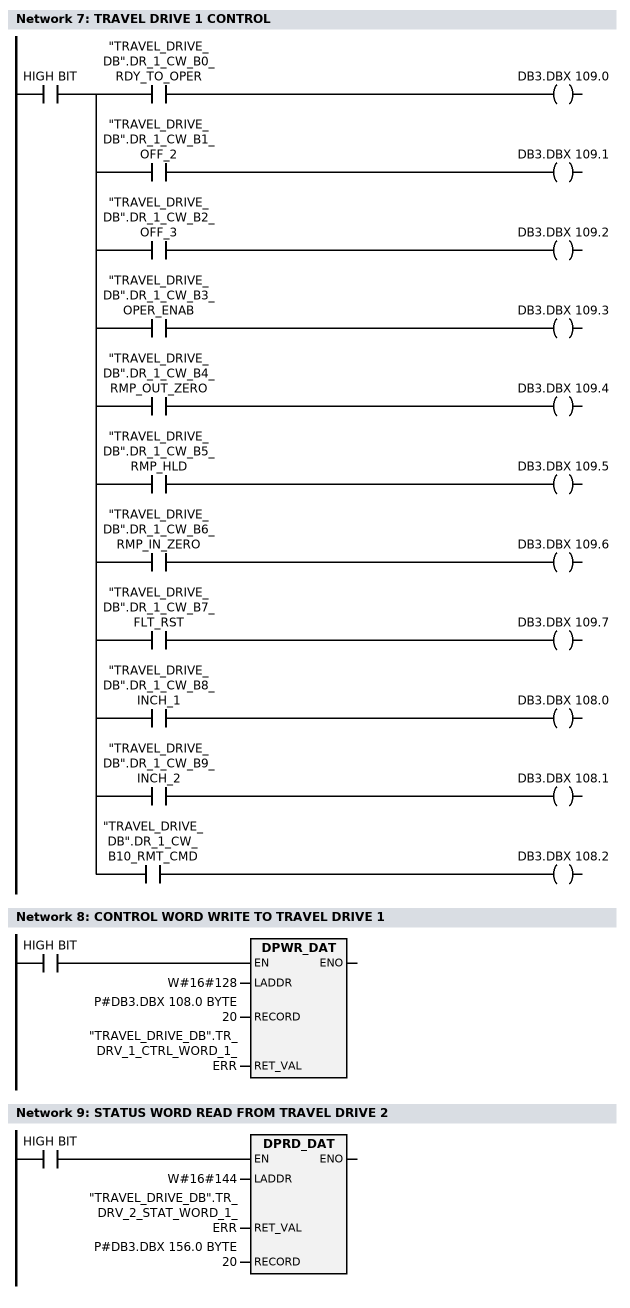
NETWORK
TITLE = TRAVEL DRIVE 1 CONTROL
      A     "HIGH BIT";
      =     L 22.0;
      A     L 22.0;
      A     "TRAVEL_DRIVE_DB".DR_1_CW_B0_RDY_TO_OPER;
      =     DB3.DBX 109.0;
      A     L 22.0;
      A     "TRAVEL_DRIVE_DB".DR_1_CW_B1_OFF_2;
      =     DB3.DBX 109.1;
      A     L 22.0;
      A     "TRAVEL_DRIVE_DB".DR_1_CW_B2_OFF_3;
      =     DB3.DBX 109.2;
      A     L 22.0;
      A     "TRAVEL_DRIVE_DB".DR_1_CW_B3_OPER_ENAB;
      =     DB3.DBX 109.3;
      A     L 22.0;
      A     "TRAVEL_DRIVE_DB".DR_1_CW_B4_RMP_OUT_ZERO;
      =     DB3.DBX 109.4;
      A     L 22.0;
      A     "TRAVEL_DRIVE_DB".DR_1_CW_B5_RMP_HLD;
      =     DB3.DBX 109.5;
      A     L 22.0;
      A     "TRAVEL_DRIVE_DB".DR_1_CW_B6_RMP_IN_ZERO;
      =     DB3.DBX 109.6;
      A     L 22.0;
      A     "TRAVEL_DRIVE_DB".DR_1_CW_B7_FLT_RST;
      =     DB3.DBX 109.7;
      A     L 22.0;
      A     "TRAVEL_DRIVE_DB".DR_1_CW_B8_INCH_1;
      =     DB3.DBX 108.0;
      A     L 22.0;
      A     "TRAVEL_DRIVE_DB".DR_1_CW_B9_INCH_2;
      =     DB3.DBX 108.1;
      A     L 22.0;
      A     "TRAVEL_DRIVE_DB".DR_1_CW_B10_RMT_CMD;
      =     DB3.DBX 108.2;
NETWORK
TITLE = CONTROL WORD WRITE TO TRAVEL DRIVE 1
      A     "HIGH BIT";
      JNB   _008;
      CALL  "DPWR_DAT" (
           LADDR                    := W#16#128,
           RECORD                   := P#DB3.DBX 108.0 BYTE 20,
           RET_VAL                  := "TRAVEL_DRIVE_DB".TR_DRV_1_CTRL_WORD_1_ERR);
_008: NOP   0;
NETWORK
TITLE = STATUS WORD READ FROM TRAVEL DRIVE 2
      A     "HIGH BIT";
      JNB   _009;
      CALL  "DPRD_DAT" (
           LADDR                    := W#16#144,
           RET_VAL                  := "TRAVEL_DRIVE_DB".TR_DRV_2_STAT_WORD_1_ERR,
           RECORD                   := P#DB3.DBX 156.0 BYTE 20);
_009: NOP   0;
